LIN {X 0,Y 347.72,Z 388.171,A -85,B 0,C 180,E1 -13726.687,E2 -13726.687} C_VEL
LIN {X 0,Y 347.741,Z 388.168,A -85,B 0,C 180,E1 -13730.174,E2 -13730.174} C_VEL
LIN {X 0,Y 347.757,Z 388.167,A -85,B 0,C 180,E1 -13732.681,E2 -13732.681} C_VEL
LIN {X 0,Y 347.743,Z 388.169,A -85,B 0,C 180,E1 -13735.958,E2 -13735.958} C_VEL
LIN {X 0,Y 347.838,Z 388.219,A -85,B 0,C 180,E1 -13739.799,E2 -13739.799} C_VEL
LIN {X 0,Y 350.158,Z 399.265,A -85,B 0,C 180,E1 -13742.833,E2 -13742.833} C_VEL
LIN {X 0,Y 351.631,Z 408.22,A -85,B 0,C 180,E1 -13745.185,E2 -13745.185} C_VEL
LIN {X 0,Y 351.614,Z 408.733,A -85,B 0,C 180,E1 -13745.302,E2 -13745.302} C_VEL
LIN {X 0,Y 355.783,Z 429.347,A -85,B 0,C 180,E1 -13746.384,E2 -13746.384} C_VEL
LIN {X 0,Y 358.162,Z 444.826,A -85,B 0,C 180,E1 -13747.086,E2 -13747.086} C_VEL
LIN {X 0,Y 359.103,Z 454.426,A -85,B 0,C 180,E1 -13747.462,E2 -13747.462} C_VEL
LIN {X 0,Y 356.443,Z 527.667,A -85,B 0,C 180,E1 -13749.403,E2 -13749.403} C_VEL
LIN {X 0,Y 355.433,Z 541.2,A -85,B 0,C 180,E1 -13749.983,E2 -13749.983} C_VEL
LIN {X 0,Y 354.327,Z 553.435,A -85,B 0,C 180,E1 -13750.748,E2 -13750.748} C_VEL
LIN {X 0,Y 353.054,Z 565.374,A -85,B 0,C 180,E1 -13751.73,E2 -13751.73} C_VEL
LIN {X 0,Y 351.787,Z 576.175,A -85,B 0,C 180,E1 -13752.864,E2 -13752.864} C_VEL
LIN {X 0,Y 350.439,Z 586.967,A -85,B 0,C 180,E1 -13754.288,E2 -13754.288} C_VEL
LIN {X 0,Y 349.396,Z 595.866,A -85,B 0,C 180,E1 -13755.737,E2 -13755.737} C_VEL
LIN {X 0,Y 348.24,Z 604.478,A -85,B 0,C 180,E1 -13757.472,E2 -13757.472} C_VEL
LIN {X 0,Y 347.356,Z 611.404,A -85,B 0,C 180,E1 -13759.215,E2 -13759.215} C_VEL
LIN {X 0,Y 346.698,Z 617.747,A -85,B 0,C 180,E1 -13761.257,E2 -13761.257} C_VEL
LIN {X 0,Y 346.364,Z 621.852,A -85,B 0,C 180,E1 -13763.009,E2 -13763.009} C_VEL
LIN {X 0,Y 346.173,Z 625.978,A -85,B 0,C 180,E1 -13765.344,E2 -13765.344} C_VEL
LIN {X 0,Y 346.146,Z 627.567,A -85,B 0,C 180,E1 -13766.509,E2 -13766.509} C_VEL
LIN {X 0,Y 346.085,Z 628.723,A -85,B 0,C 180,E1 -13767.674,E2 -13767.674} C_VEL
LIN {X 0,Y 346.118,Z 629.437,A -85,B 0,C 180,E1 -13768.838,E2 -13768.838} C_VEL
LIN {X 0,Y 346.164,Z 629.755,A -85,B 0,C 180,E1 -13770.002,E2 -13770.002} C_VEL
LIN {X 0,Y 346.103,Z 629.676,A -85,B 0,C 180,E1 -13771.165,E2 -13771.165} C_VEL
LIN {X 0,Y 346.083,Z 629.185,A -85,B 0,C 180,E1 -13772.329,E2 -13772.329} C_VEL
LIN {X 0,Y 346.142,Z 628.26,A -85,B 0,C 180,E1 -13773.494,E2 -13773.494} C_VEL
LIN {X 0,Y 346.161,Z 626.933,A -85,B 0,C 180,E1 -13774.66,E2 -13774.66} C_VEL
LIN {X 0,Y 346.261,Z 624.135,A -85,B 0,C 180,E1 -13776.41,E2 -13776.41} C_VEL
LIN {X 0,Y 346.568,Z 620.305,A -85,B 0,C 180,E1 -13778.162,E2 -13778.162} C_VEL
LIN {X 0,Y 347.043,Z 615.354,A -85,B 0,C 180,E1 -13779.913,E2 -13779.913} C_VEL
LIN {X 0,Y 347.727,Z 609.133,A -85,B 0,C 180,E1 -13781.662,E2 -13781.662} C_VEL
LIN {X 0,Y 348.808,Z 601.409,A -85,B 0,C 180,E1 -13783.399,E2 -13783.399} C_VEL
LIN {X 0,Y 349.843,Z 593.517,A -85,B 0,C 180,E1 -13784.842,E2 -13784.842} C_VEL
LIN {X 0,Y 350.944,Z 583.905,A -85,B 0,C 180,E1 -13786.283,E2 -13786.283} C_VEL
LIN {X 0,Y 352.227,Z 573.271,A -85,B 0,C 180,E1 -13787.567,E2 -13787.567} C_VEL
LIN {X 0,Y 353.609,Z 561.389,A -85,B 0,C 180,E1 -13788.694,E2 -13788.694} C_VEL
LIN {X 0,Y 354.715,Z 548.741,A -85,B 0,C 180,E1 -13789.609,E2 -13789.609} C_VEL
LIN {X 0,Y 355.742,Z 536.184,A -85,B 0,C 180,E1 -13790.265,E2 -13790.265} C_VEL
LIN {X 0,Y 356.474,Z 523.056,A -85,B 0,C 180,E1 -13790.712,E2 -13790.712} C_VEL
LIN {X 0,Y 357.988,Z 452.327,A -85,B 0,C 180,E1 -13792.264,E2 -13792.264} C_VEL
LIN {X 0,Y 354.472,Z 430.592,A -85,B 0,C 180,E1 -13793.053,E2 -13793.053} C_VEL
LIN {X 0,Y 351.716,Z 416.728,A -85,B 0,C 180,E1 -13793.635,E2 -13793.635} C_VEL
LIN {X 0,Y 352.39,Z 410.952,A -85,B 0,C 180,E1 -13795.077,E2 -13795.077} C_VEL
LIN {X 0,Y 351.496,Z 404.927,A -85,B 0,C 180,E1 -13796.737,E2 -13796.737} C_VEL
LIN {X 0,Y 349.55,Z 395.513,A -85,B 0,C 180,E1 -13799.471,E2 -13799.471} C_VEL
LIN {X 0,Y 347.759,Z 388.171,A -85,B 0,C 180,E1 -13801.755,E2 -13801.755} C_VEL
LIN {X 0,Y 347.794,Z 388.165,A -85,B 0,C 180,E1 -13805.876,E2 -13805.876} C_VEL
LIN {X 0,Y 347.757,Z 388.171,A -85,B 0,C 180,E1 -13808.793,E2 -13808.793} C_VEL
LIN {X 0,Y 347.756,Z 388.17,A -85,B 0,C 180,E1 -13811.831,E2 -13811.831} C_VEL
LIN {X 0,Y 347.711,Z 388.173,A -85,B 0,C 180,E1 -13815.027,E2 -13815.027} C_VEL
LIN {X 0,Y 347.756,Z 388.167,A -85,B 0,C 180,E1 -13818.398,E2 -13818.398} C_VEL
LIN {X 0,Y 347.779,Z 388.163,A -85,B 0,C 180,E1 -13822.012,E2 -13822.012} C_VEL
LIN {X 0,Y 347.75,Z 388.163,A -85,B 0,C 180,E1 -13825.537,E2 -13825.537} C_VEL
LIN {X 0,Y 347.751,Z 388.168,A -85,B 0,C 180,E1 -13828.301,E2 -13828.301} C_VEL
LIN {X 0,Y 347.785,Z 388.164,A -85,B 0,C 180,E1 -13830.988,E2 -13830.988} C_VEL
LIN {X 0,Y 347.837,Z 388.149,A -85,B 0,C 180,E1 -13833.608,E2 -13833.608} C_VEL
LIN {X 0,Y 347.795,Z 388.162,A -85,B 0,C 180,E1 -13836.162,E2 -13836.162} C_VEL
LIN {X 0,Y 347.819,Z 388.159,A -85,B 0,C 180,E1 -13839.91,E2 -13839.91} C_VEL
LIN {X 0,Y 347.873,Z 388.148,A -85,B 0,C 180,E1 -13842.36,E2 -13842.36} C_VEL
LIN {X 0,Y 347.904,Z 388.14,A -85,B 0,C 180,E1 -13845.971,E2 -13845.971} C_VEL
LIN {X 0,Y 347.935,Z 388.136,A -85,B 0,C 180,E1 -13849.526,E2 -13849.526} C_VEL
LIN {X 0,Y 348.081,Z 388.128,A -85,B 0,C 180,E1 -13851.875,E2 -13851.875} C_VEL
LIN {X 0,Y 348.074,Z 388.123,A -85,B 0,C 180,E1 -13854.206,E2 -13854.206} C_VEL
LIN {X 0,Y 348.212,Z 388.103,A -85,B 0,C 180,E1 -13857.687,E2 -13857.687} C_VEL
LIN {X 0,Y 348.332,Z 388.092,A -85,B 0,C 180,E1 -13860,E2 -13860} C_VEL
LIN {X 0,Y 348.213,Z 388.111,A -85,B 0,C 180,E1 -13862.314,E2 -13862.314} C_VEL
LIN {X 0,Y 348.113,Z 388.118,A -85,B 0,C 180,E1 -13866.958,E2 -13866.958} C_VEL
LIN {X 0,Y 347.974,Z 388.139,A -85,B 0,C 180,E1 -13869.298,E2 -13869.298} C_VEL
LIN {X 0,Y 347.897,Z 388.149,A -85,B 0,C 180,E1 -13872.839,E2 -13872.839} C_VEL
LIN {X 0,Y 347.846,Z 388.157,A -85,B 0,C 180,E1 -13876.431,E2 -13876.431} C_VEL
LIN {X 0,Y 347.863,Z 388.156,A -85,B 0,C 180,E1 -13878.86,E2 -13878.86} C_VEL
LIN {X 0,Y 347.781,Z 388.166,A -85,B 0,C 180,E1 -13882.579,E2 -13882.579} C_VEL
LIN {X 0,Y 347.829,Z 388.166,A -85,B 0,C 180,E1 -13884.238,E2 -13884.238} C_VEL
LIN {X 0,Y 350.024,Z 397.889,A -85,B 0,C 180,E1 -13887.504,E2 -13887.504} C_VEL
LIN {X 0,Y 350.495,Z 400.533,A -85,B 0,C 180,E1 -13888.353,E2 -13888.353} C_VEL
LIN {X 0,Y 355.561,Z 413.584,A -85,B 0,C 180,E1 -13889.086,E2 -13889.086} C_VEL
LIN {X 0,Y 358.59,Z 428.221,A -85,B 0,C 180,E1 -13889.672,E2 -13889.672} C_VEL
LIN {X 0,Y 356.597,Z 507.412,A -85,B 0,C 180,E1 -13891.413,E2 -13891.413} C_VEL
LIN {X 0,Y 355.951,Z 520.049,A -85,B 0,C 180,E1 -13891.895,E2 -13891.895} C_VEL
LIN {X 0,Y 355.055,Z 533.276,A -85,B 0,C 180,E1 -13892.642,E2 -13892.642} C_VEL
LIN {X 0,Y 353.946,Z 545.604,A -85,B 0,C 180,E1 -13893.604,E2 -13893.604} C_VEL
LIN {X 0,Y 352.773,Z 556.709,A -85,B 0,C 180,E1 -13894.721,E2 -13894.721} C_VEL
LIN {X 0,Y 351.601,Z 566.56,A -85,B 0,C 180,E1 -13895.956,E2 -13895.956} C_VEL
LIN {X 0,Y 350.493,Z 575.046,A -85,B 0,C 180,E1 -13897.256,E2 -13897.256} C_VEL
LIN {X 0,Y 349.382,Z 583.6,A -85,B 0,C 180,E1 -13898.868,E2 -13898.868} C_VEL
LIN {X 0,Y 348.401,Z 590.791,A -85,B 0,C 180,E1 -13900.543,E2 -13900.543} C_VEL
LIN {X 0,Y 347.524,Z 597.568,A -85,B 0,C 180,E1 -13902.536,E2 -13902.536} C_VEL
LIN {X 0,Y 346.932,Z 601.844,A -85,B 0,C 180,E1 -13904.154,E2 -13904.154} C_VEL
LIN {X 0,Y 346.562,Z 605.2,A -85,B 0,C 180,E1 -13905.792,E2 -13905.792} C_VEL
LIN {X 0,Y 346.141,Z 608.29,A -85,B 0,C 180,E1 -13907.929,E2 -13907.929} C_VEL
LIN {X 0,Y 345.978,Z 609.589,A -85,B 0,C 180,E1 -13909.455,E2 -13909.455} C_VEL
LIN {X 0,Y 345.904,Z 610.218,A -85,B 0,C 180,E1 -13910.959,E2 -13910.959} C_VEL
LIN {X 0,Y 345.879,Z 610.181,A -85,B 0,C 180,E1 -13912.44,E2 -13912.44} C_VEL
LIN {X 0,Y 345.94,Z 609.166,A -85,B 0,C 180,E1 -13914.354,E2 -13914.354} C_VEL
LIN {X 0,Y 346.175,Z 606.93,A -85,B 0,C 180,E1 -13916.344,E2 -13916.344} C_VEL
LIN {X 0,Y 346.537,Z 603.249,A -85,B 0,C 180,E1 -13918.407,E2 -13918.407} C_VEL
LIN {X 0,Y 346.857,Z 599.121,A -85,B 0,C 180,E1 -13920.107,E2 -13920.107} C_VEL
LIN {X 0,Y 347.444,Z 593.365,A -85,B 0,C 180,E1 -13921.945,E2 -13921.945} C_VEL
LIN {X 0,Y 348.176,Z 586.714,A -85,B 0,C 180,E1 -13923.634,E2 -13923.634} C_VEL
LIN {X 0,Y 349.022,Z 578.446,A -85,B 0,C 180,E1 -13925.33,E2 -13925.33} C_VEL
LIN {X 0,Y 350.071,Z 569.169,A -85,B 0,C 180,E1 -13926.851,E2 -13926.851} C_VEL
LIN {X 0,Y 351.212,Z 558.436,A -85,B 0,C 180,E1 -13928.271,E2 -13928.271} C_VEL
LIN {X 0,Y 352.121,Z 547.542,A -85,B 0,C 180,E1 -13929.422,E2 -13929.422} C_VEL
LIN {X 0,Y 353.153,Z 534.893,A -85,B 0,C 180,E1 -13930.452,E2 -13930.452} C_VEL
LIN {X 0,Y 353.886,Z 523.166,A -85,B 0,C 180,E1 -13931.171,E2 -13931.171} C_VEL
LIN {X 0,Y 354.534,Z 510.132,A -85,B 0,C 180,E1 -13931.726,E2 -13931.726} C_VEL
LIN {X 0,Y 354.958,Z 492.695,A -85,B 0,C 180,E1 -13932.16,E2 -13932.16} C_VEL
LIN {X 0,Y 356.276,Z 426.34,A -85,B 0,C 180,E1 -13933.571,E2 -13933.571} C_VEL
LIN {X 0,Y 352.164,Z 405.889,A -85,B 0,C 180,E1 -13934.276,E2 -13934.276} C_VEL
LIN {X 0,Y 350.017,Z 399.405,A -85,B 0,C 180,E1 -13934.569,E2 -13934.569} C_VEL
LIN {X 0,Y 347.928,Z 388.186,A -85,B 0,C 180,E1 -13937.938,E2 -13937.938} C_VEL
LIN {X 0,Y 348.027,Z 388.131,A -85,B 0,C 180,E1 -13941.872,E2 -13941.872} C_VEL
LIN {X 0,Y 348.055,Z 388.13,A -85,B 0,C 180,E1 -13944.204,E2 -13944.204} C_VEL
LIN {X 0,Y 348.21,Z 388.108,A -85,B 0,C 180,E1 -13947.685,E2 -13947.685} C_VEL
LIN {X 0,Y 348.348,Z 388.093,A -85,B 0,C 180,E1 -13949.998,E2 -13949.998} C_VEL
LIN {X 0,Y 348.211,Z 388.113,A -85,B 0,C 180,E1 -13952.312,E2 -13952.312} C_VEL
LIN {X 0,Y 348.109,Z 388.12,A -85,B 0,C 180,E1 -13956.956,E2 -13956.956} C_VEL
LIN {X 0,Y 347.969,Z 388.137,A -85,B 0,C 180,E1 -13959.297,E2 -13959.297} C_VEL
LIN {X 0,Y 347.891,Z 388.147,A -85,B 0,C 180,E1 -13962.838,E2 -13962.838} C_VEL
LIN {X 0,Y 347.842,Z 388.155,A -85,B 0,C 180,E1 -13966.43,E2 -13966.43} C_VEL
LIN {X 0,Y 347.817,Z 388.156,A -85,B 0,C 180,E1 -13969.381,E2 -13969.381} C_VEL
LIN {X 0,Y 347.123,Z 388.247,A -85,B 0,C 180,E1 -13970.346,E2 -13970.346} C_VEL
LIN {X 0,Y 344.256,Z 388.606,A -85,B 0,C 180,E1 -13971.917,E2 -13971.917} C_VEL
LIN {X 0,Y 341.85,Z 388.905,A -85,B 0,C 180,E1 -13973.188,E2 -13973.188} C_VEL
LIN {X 0,Y 340.83,Z 389.03,A -85,B 0,C 180,E1 -13974.172,E2 -13974.172} C_VEL
LIN {X 0,Y 340.753,Z 389.037,A -85,B 0,C 180,E1 -13974.505,E2 -13974.505} C_VEL
LIN {X 0,Y 340.778,Z 389.036,A -85,B 0,C 180,E1 -13977.525,E2 -13977.525} C_VEL
LIN {X 0,Y 340.714,Z 389.041,A -85,B 0,C 180,E1 -13981.041,E2 -13981.041} C_VEL
LIN {X 0,Y 340.715,Z 389.043,A -85,B 0,C 180,E1 -13985.277,E2 -13985.277} C_VEL
LIN {X 0,Y 340.715,Z 389.041,A -85,B 0,C 180,E1 -13988.386,E2 -13988.386} C_VEL
LIN {X 0,Y 340.728,Z 389.041,A -85,B 0,C 180,E1 -13992.05,E2 -13992.05} C_VEL
LIN {X 0,Y 340.751,Z 389.142,A -85,B 0,C 180,E1 -13993.651,E2 -13993.651} C_VEL
LIN {X 0,Y 342.514,Z 397.857,A -85,B 0,C 180,E1 -13995.733,E2 -13995.733} C_VEL
LIN {X 0,Y 344.996,Z 407.303,A -85,B 0,C 180,E1 -13996.109,E2 -13996.109} C_VEL
LIN {X 0,Y 348.332,Z 426.928,A -85,B 0,C 180,E1 -13996.786,E2 -13996.786} C_VEL
LIN {X 0,Y 346.221,Z 507.298,A -85,B 0,C 180,E1 -13998.782,E2 -13998.782} C_VEL
LIN {X 0,Y 345.703,Z 520.636,A -85,B 0,C 180,E1 -13999.342,E2 -13999.342} C_VEL
LIN {X 0,Y 344.889,Z 534.013,A -85,B 0,C 180,E1 -14000.162,E2 -14000.162} C_VEL
LIN {X 0,Y 344.107,Z 545.469,A -85,B 0,C 180,E1 -14001.094,E2 -14001.094} C_VEL
LIN {X 0,Y 343.207,Z 556.587,A -85,B 0,C 180,E1 -14002.25,E2 -14002.25} C_VEL
LIN {X 0,Y 342.276,Z 567.32,A -85,B 0,C 180,E1 -14003.637,E2 -14003.637} C_VEL
LIN {X 0,Y 341.384,Z 576.974,A -85,B 0,C 180,E1 -14005.193,E2 -14005.193} C_VEL
LIN {X 0,Y 340.642,Z 585.34,A -85,B 0,C 180,E1 -14006.856,E2 -14006.856} C_VEL
LIN {X 0,Y 340.115,Z 591.566,A -85,B 0,C 180,E1 -14008.37,E2 -14008.37} C_VEL
LIN {X 0,Y 339.565,Z 598.161,A -85,B 0,C 180,E1 -14010.371,E2 -14010.371} C_VEL
LIN {X 0,Y 339.29,Z 602.813,A -85,B 0,C 180,E1 -14012.221,E2 -14012.221} C_VEL
LIN {X 0,Y 338.978,Z 606.451,A -85,B 0,C 180,E1 -14014.19,E2 -14014.19} C_VEL
LIN {X 0,Y 338.841,Z 608.553,A -85,B 0,C 180,E1 -14015.865,E2 -14015.865} C_VEL
LIN {X 0,Y 338.75,Z 610.039,A -85,B 0,C 180,E1 -14018.072,E2 -14018.072} C_VEL
LIN {X 0,Y 338.843,Z 610.196,A -85,B 0,C 180,E1 -14019.353,E2 -14019.353} C_VEL
LIN {X 0,Y 338.914,Z 609.887,A -85,B 0,C 180,E1 -14020.622,E2 -14020.622} C_VEL
LIN {X 0,Y 339.179,Z 608.649,A -85,B 0,C 180,E1 -14022.385,E2 -14022.385} C_VEL
LIN {X 0,Y 339.511,Z 606.116,A -85,B 0,C 180,E1 -14024.389,E2 -14024.389} C_VEL
LIN {X 0,Y 340.001,Z 602.542,A -85,B 0,C 180,E1 -14026.283,E2 -14026.283} C_VEL
LIN {X 0,Y 340.778,Z 597.891,A -85,B 0,C 180,E1 -14028.098,E2 -14028.098} C_VEL
LIN {X 0,Y 341.689,Z 591.642,A -85,B 0,C 180,E1 -14029.991,E2 -14029.991} C_VEL
LIN {X 0,Y 342.831,Z 584.319,A -85,B 0,C 180,E1 -14031.749,E2 -14031.749} C_VEL
LIN {X 0,Y 344.018,Z 576.597,A -85,B 0,C 180,E1 -14033.254,E2 -14033.254} C_VEL
LIN {X 0,Y 345.367,Z 566.981,A -85,B 0,C 180,E1 -14034.775,E2 -14034.775} C_VEL
LIN {X 0,Y 346.799,Z 556.812,A -85,B 0,C 180,E1 -14036.078,E2 -14036.078} C_VEL
LIN {X 0,Y 348.151,Z 545.387,A -85,B 0,C 180,E1 -14037.252,E2 -14037.252} C_VEL
LIN {X 0,Y 349.395,Z 532.56,A -85,B 0,C 180,E1 -14038.271,E2 -14038.271} C_VEL
LIN {X 0,Y 350.408,Z 519.533,A -85,B 0,C 180,E1 -14039.03,E2 -14039.03} C_VEL
LIN {X 0,Y 351.237,Z 505.365,A -85,B 0,C 180,E1 -14039.585,E2 -14039.585} C_VEL
LIN {X 0,Y 354.285,Z 429.068,A -85,B 0,C 180,E1 -14041.595,E2 -14041.595} C_VEL
LIN {X 0,Y 351.519,Z 416.043,A -85,B 0,C 180,E1 -14042.292,E2 -14042.292} C_VEL
LIN {X 0,Y 346.855,Z 405.479,A -85,B 0,C 180,E1 -14043.142,E2 -14043.142} C_VEL
LIN {X 0,Y 343.776,Z 399.199,A -85,B 0,C 180,E1 -14043.736,E2 -14043.736} C_VEL
LIN {X 0,Y 341.037,Z 389.005,A -85,B 0,C 180,E1 -14046.619,E2 -14046.619} C_VEL
LIN {X 0,Y 340.919,Z 389.02,A -85,B 0,C 180,E1 -14049.492,E2 -14049.492} C_VEL
LIN {X 0,Y 340.836,Z 389.031,A -85,B 0,C 180,E1 -14053.11,E2 -14053.11} C_VEL
LIN {X 0,Y 340.778,Z 389.037,A -85,B 0,C 180,E1 -14056.782,E2 -14056.782} C_VEL
LIN {X 0,Y 340.796,Z 389.035,A -85,B 0,C 180,E1 -14059.266,E2 -14059.266} C_VEL
LIN {X 0,Y 340.767,Z 389.036,A -85,B 0,C 180,E1 -14063.07,E2 -14063.07} C_VEL
LIN {X 0,Y 340.796,Z 389.034,A -85,B 0,C 180,E1 -14066.981,E2 -14066.981} C_VEL
LIN {X 0,Y 340.756,Z 389.039,A -85,B 0,C 180,E1 -14069.98,E2 -14069.98} C_VEL
LIN {X 0,Y 340.686,Z 389.048,A -85,B 0,C 180,E1 -14073.847,E2 -14073.847} C_VEL
LIN {X 0,Y 340.699,Z 389.046,A -85,B 0,C 180,E1 -14076.742,E2 -14076.742} C_VEL
LIN {X 0,Y 340.681,Z 389.048,A -85,B 0,C 180,E1 -14080.248,E2 -14080.248} C_VEL
LIN {X 0,Y 340.66,Z 389.05,A -85,B 0,C 180,E1 -14083.777,E2 -14083.777} C_VEL
LIN {X 0,Y 340.67,Z 389.051,A -85,B 0,C 180,E1 -14087.097,E2 -14087.097} C_VEL
LIN {X 0,Y 340.693,Z 389.047,A -85,B 0,C 180,E1 -14090.249,E2 -14090.249} C_VEL
LIN {X 0,Y 340.705,Z 389.044,A -85,B 0,C 180,E1 -14093.561,E2 -14093.561} C_VEL
LIN {X 0,Y 340.691,Z 389.048,A -85,B 0,C 180,E1 -14096.155,E2 -14096.155} C_VEL
LIN {X 0,Y 340.773,Z 389.154,A -85,B 0,C 180,E1 -14099.486,E2 -14099.486} C_VEL
LIN {X 0,Y 343.37,Z 401.381,A -85,B 0,C 180,E1 -14102.911,E2 -14102.911} C_VEL
LIN {X 0,Y 344.42,Z 407.215,A -85,B 0,C 180,E1 -14104.447,E2 -14104.447} C_VEL
LIN {X 0,Y 346.267,Z 413.478,A -85,B 0,C 180,E1 -14104.87,E2 -14104.87} C_VEL
LIN {X 0,Y 349.592,Z 430.004,A -85,B 0,C 180,E1 -14105.772,E2 -14105.772} C_VEL
LIN {X 0,Y 351.931,Z 445.044,A -85,B 0,C 180,E1 -14106.5,E2 -14106.5} C_VEL
LIN {X 0,Y 352.925,Z 455.244,A -85,B 0,C 180,E1 -14106.913,E2 -14106.913} C_VEL
LIN {X 0,Y 350.131,Z 526.949,A -85,B 0,C 180,E1 -14108.86,E2 -14108.86} C_VEL
LIN {X 0,Y 349.095,Z 540.506,A -85,B 0,C 180,E1 -14109.45,E2 -14109.45} C_VEL
LIN {X 0,Y 347.924,Z 552.831,A -85,B 0,C 180,E1 -14110.226,E2 -14110.226} C_VEL
LIN {X 0,Y 346.562,Z 564.849,A -85,B 0,C 180,E1 -14111.222,E2 -14111.222} C_VEL
LIN {X 0,Y 345.243,Z 575.728,A -85,B 0,C 180,E1 -14112.376,E2 -14112.376} C_VEL
LIN {X 0,Y 343.733,Z 586.753,A -85,B 0,C 180,E1 -14113.851,E2 -14113.851} C_VEL
LIN {X 0,Y 342.531,Z 596.263,A -85,B 0,C 180,E1 -14115.445,E2 -14115.445} C_VEL
LIN {X 0,Y 341.303,Z 604.719,A -85,B 0,C 180,E1 -14117.213,E2 -14117.213} C_VEL
LIN {X 0,Y 340.377,Z 611.576,A -85,B 0,C 180,E1 -14118.991,E2 -14118.991} C_VEL
LIN {X 0,Y 339.663,Z 617.816,A -85,B 0,C 180,E1 -14121.074,E2 -14121.074} C_VEL
LIN {X 0,Y 339.311,Z 621.854,A -85,B 0,C 180,E1 -14122.863,E2 -14122.863} C_VEL
LIN {X 0,Y 339.078,Z 625.706,A -85,B 0,C 180,E1 -14125.246,E2 -14125.246} C_VEL
LIN {X 0,Y 339.07,Z 627.31,A -85,B 0,C 180,E1 -14126.437,E2 -14126.437} C_VEL
LIN {X 0,Y 338.999,Z 628.489,A -85,B 0,C 180,E1 -14127.625,E2 -14127.625} C_VEL
LIN {X 0,Y 339.02,Z 629.217,A -85,B 0,C 180,E1 -14128.814,E2 -14128.814} C_VEL
LIN {X 0,Y 339.067,Z 629.547,A -85,B 0,C 180,E1 -14130.002,E2 -14130.002} C_VEL
LIN {X 0,Y 339.006,Z 629.48,A -85,B 0,C 180,E1 -14131.189,E2 -14131.189} C_VEL
LIN {X 0,Y 338.998,Z 629.011,A -85,B 0,C 180,E1 -14132.378,E2 -14132.378} C_VEL
LIN {X 0,Y 339.066,Z 628.1,A -85,B 0,C 180,E1 -14133.567,E2 -14133.567} C_VEL
LIN {X 0,Y 339.112,Z 625.216,A -85,B 0,C 180,E1 -14135.852,E2 -14135.852} C_VEL
LIN {X 0,Y 339.401,Z 621.617,A -85,B 0,C 180,E1 -14137.737,E2 -14137.737} C_VEL
LIN {X 0,Y 339.827,Z 617.086,A -85,B 0,C 180,E1 -14139.525,E2 -14139.525} C_VEL
LIN {X 0,Y 340.511,Z 611.351,A -85,B 0,C 180,E1 -14141.309,E2 -14141.309} C_VEL
LIN {X 0,Y 341.525,Z 604.174,A -85,B 0,C 180,E1 -14143.084,E2 -14143.084} C_VEL
LIN {X 0,Y 342.761,Z 595.245,A -85,B 0,C 180,E1 -14144.852,E2 -14144.852} C_VEL
LIN {X 0,Y 343.995,Z 585.259,A -85,B 0,C 180,E1 -14146.447,E2 -14146.447} C_VEL
LIN {X 0,Y 345.339,Z 574.762,A -85,B 0,C 180,E1 -14147.776,E2 -14147.776} C_VEL
LIN {X 0,Y 346.737,Z 563.351,A -85,B 0,C 180,E1 -14148.925,E2 -14148.925} C_VEL
LIN {X 0,Y 347.932,Z 551.525,A -85,B 0,C 180,E1 -14149.854,E2 -14149.854} C_VEL
LIN {X 0,Y 348.999,Z 538.551,A -85,B 0,C 180,E1 -14150.598,E2 -14150.598} C_VEL
LIN {X 0,Y 349.908,Z 524.861,A -85,B 0,C 180,E1 -14151.119,E2 -14151.119} C_VEL
LIN {X 0,Y 351.573,Z 453.595,A -85,B 0,C 180,E1 -14152.724,E2 -14152.724} C_VEL
LIN {X 0,Y 348.302,Z 432.882,A -85,B 0,C 180,E1 -14153.491,E2 -14153.491} C_VEL
LIN {X 0,Y 345,Z 416.504,A -85,B 0,C 180,E1 -14154.204,E2 -14154.204} C_VEL
LIN {X 0,Y 345.509,Z 412.267,A -85,B 0,C 180,E1 -14155.289,E2 -14155.289} C_VEL
LIN {X 0,Y 344.128,Z 403.871,A -85,B 0,C 180,E1 -14157.687,E2 -14157.687} C_VEL
LIN {X 0,Y 342.167,Z 394.993,A -85,B 0,C 180,E1 -14160.382,E2 -14160.382} C_VEL
LIN {X 0,Y 340.684,Z 389.052,A -85,B 0,C 180,E1 -14162.325,E2 -14162.325} C_VEL
LIN {X 0,Y 340.723,Z 389.044,A -85,B 0,C 180,E1 -14165.28,E2 -14165.28} C_VEL
LIN {X 0,Y 340.715,Z 389.047,A -85,B 0,C 180,E1 -14168.387,E2 -14168.387} C_VEL
LIN {X 0,Y 340.704,Z 389.048,A -85,B 0,C 180,E1 -14172.046,E2 -14172.046} C_VEL
LIN {X 0,Y 340.657,Z 389.053,A -85,B 0,C 180,E1 -14176.228,E2 -14176.228} C_VEL
LIN {X 0,Y 340.693,Z 389.041,A -85,B 0,C 180,E1 -14179.754,E2 -14179.754} C_VEL
LIN {X 0,Y 340.71,Z 389.041,A -85,B 0,C 180,E1 -14183.259,E2 -14183.259} C_VEL
LIN {X 0,Y 340.698,Z 389.04,A -85,B 0,C 180,E1 -14186.154,E2 -14186.154} C_VEL
LIN {X 0,Y 340.747,Z 389.033,A -85,B 0,C 180,E1 -14190.33,E2 -14190.33} C_VEL
LIN {X 0,Y 340.809,Z 389.024,A -85,B 0,C 180,E1 -14193.02,E2 -14193.02} C_VEL
LIN {X 0,Y 340.762,Z 389.037,A -85,B 0,C 180,E1 -14195.639,E2 -14195.639} C_VEL
LIN {X 0,Y 340.759,Z 389.037,A -85,B 0,C 180,E1 -14199.475,E2 -14199.475} C_VEL
LIN {X 0,Y 340.864,Z 389.017,A -85,B 0,C 180,E1 -14201.985,E2 -14201.985} C_VEL
LIN {X 0,Y 340.876,Z 389.014,A -85,B 0,C 180,E1 -14205.705,E2 -14205.705} C_VEL
LIN {X 0,Y 340.877,Z 389.015,A -85,B 0,C 180,E1 -14209.306,E2 -14209.306} C_VEL
LIN {X 0,Y 341.082,Z 388.991,A -85,B 0,C 180,E1 -14212.898,E2 -14212.898} C_VEL
LIN {X 0,Y 341.174,Z 388.98,A -85,B 0,C 180,E1 -14217.639,E2 -14217.639} C_VEL
LIN {X 0,Y 341.282,Z 388.97,A -85,B 0,C 180,E1 -14220,E2 -14220} C_VEL
LIN {X 0,Y 341.174,Z 388.987,A -85,B 0,C 180,E1 -14222.361,E2 -14222.361} C_VEL
LIN {X 0,Y 341.082,Z 388.994,A -85,B 0,C 180,E1 -14227.102,E2 -14227.102} C_VEL
LIN {X 0,Y 340.878,Z 389.025,A -85,B 0,C 180,E1 -14230.694,E2 -14230.694} C_VEL
LIN {X 0,Y 340.87,Z 389.024,A -85,B 0,C 180,E1 -14234.325,E2 -14234.325} C_VEL
LIN {X 0,Y 340.845,Z 389.03,A -85,B 0,C 180,E1 -14238.467,E2 -14238.467} C_VEL
LIN {X 0,Y 340.761,Z 389.04,A -85,B 0,C 180,E1 -14241.857,E2 -14241.857} C_VEL
LIN {X 0,Y 340.757,Z 389.053,A -85,B 0,C 180,E1 -14243.715,E2 -14243.715} C_VEL
LIN {X 0,Y 342.797,Z 397.988,A -85,B 0,C 180,E1 -14246.811,E2 -14246.811} C_VEL
LIN {X 0,Y 343.412,Z 400.853,A -85,B 0,C 180,E1 -14247.748,E2 -14247.748} C_VEL
LIN {X 0,Y 349.277,Z 415.294,A -85,B 0,C 180,E1 -14248.619,E2 -14248.619} C_VEL
LIN {X 0,Y 352.168,Z 429.023,A -85,B 0,C 180,E1 -14249.189,E2 -14249.189} C_VEL
LIN {X 0,Y 350.081,Z 508.162,A -85,B 0,C 180,E1 -14250.969,E2 -14250.969} C_VEL
LIN {X 0,Y 349.405,Z 520.702,A -85,B 0,C 180,E1 -14251.464,E2 -14251.464} C_VEL
LIN {X 0,Y 348.563,Z 532.323,A -85,B 0,C 180,E1 -14252.129,E2 -14252.129} C_VEL
LIN {X 0,Y 347.565,Z 543.421,A -85,B 0,C 180,E1 -14252.971,E2 -14252.971} C_VEL
LIN {X 0,Y 346.416,Z 554.353,A -85,B 0,C 180,E1 -14254.036,E2 -14254.036} C_VEL
LIN {X 0,Y 345.256,Z 563.645,A -85,B 0,C 180,E1 -14255.155,E2 -14255.155} C_VEL
LIN {X 0,Y 343.903,Z 573.946,A -85,B 0,C 180,E1 -14256.693,E2 -14256.693} C_VEL
LIN {X 0,Y 342.617,Z 582.852,A -85,B 0,C 180,E1 -14258.342,E2 -14258.342} C_VEL
LIN {X 0,Y 341.565,Z 590.039,A -85,B 0,C 180,E1 -14259.998,E2 -14259.998} C_VEL
LIN {X 0,Y 340.595,Z 596.982,A -85,B 0,C 180,E1 -14262.024,E2 -14262.024} C_VEL
LIN {X 0,Y 339.84,Z 602.692,A -85,B 0,C 180,E1 -14264.219,E2 -14264.219} C_VEL
LIN {X 0,Y 339.306,Z 606.782,A -85,B 0,C 180,E1 -14266.465,E2 -14266.465} C_VEL
LIN {X 0,Y 339.017,Z 609.108,A -85,B 0,C 180,E1 -14268.441,E2 -14268.441} C_VEL
LIN {X 0,Y 338.827,Z 610.191,A -85,B 0,C 180,E1 -14270.127,E2 -14270.127} C_VEL
LIN {X 0,Y 338.757,Z 610.441,A -85,B 0,C 180,E1 -14272.033,E2 -14272.033} C_VEL
LIN {X 0,Y 338.832,Z 609.619,A -85,B 0,C 180,E1 -14273.992,E2 -14273.992} C_VEL
LIN {X 0,Y 339.028,Z 607.609,A -85,B 0,C 180,E1 -14276.017,E2 -14276.017} C_VEL
LIN {X 0,Y 339.394,Z 604.249,A -85,B 0,C 180,E1 -14278.104,E2 -14278.104} C_VEL
LIN {X 0,Y 339.826,Z 599.117,A -85,B 0,C 180,E1 -14280.298,E2 -14280.298} C_VEL
LIN {X 0,Y 340.428,Z 593.459,A -85,B 0,C 180,E1 -14282.13,E2 -14282.13} C_VEL
LIN {X 0,Y 341.283,Z 585.953,A -85,B 0,C 180,E1 -14284.048,E2 -14284.048} C_VEL
LIN {X 0,Y 342.178,Z 577.564,A -85,B 0,C 180,E1 -14285.745,E2 -14285.745} C_VEL
LIN {X 0,Y 343.254,Z 568.286,A -85,B 0,C 180,E1 -14287.263,E2 -14287.263} C_VEL
LIN {X 0,Y 344.355,Z 558.306,A -85,B 0,C 180,E1 -14288.588,E2 -14288.588} C_VEL
LIN {X 0,Y 345.305,Z 547.35,A -85,B 0,C 180,E1 -14289.756,E2 -14289.756} C_VEL
LIN {X 0,Y 346.302,Z 535.448,A -85,B 0,C 180,E1 -14290.743,E2 -14290.743} C_VEL
LIN {X 0,Y 347.123,Z 522.735,A -85,B 0,C 180,E1 -14291.537,E2 -14291.537} C_VEL
LIN {X 0,Y 347.776,Z 509.585,A -85,B 0,C 180,E1 -14292.092,E2 -14292.092} C_VEL
LIN {X 0,Y 348.242,Z 489.439,A -85,B 0,C 180,E1 -14292.587,E2 -14292.587} C_VEL
LIN {X 0,Y 349.556,Z 427.119,A -85,B 0,C 180,E1 -14293.941,E2 -14293.941} C_VEL
LIN {X 0,Y 345.605,Z 407.6,A -85,B 0,C 180,E1 -14294.631,E2 -14294.631} C_VEL
LIN {X 0,Y 342.873,Z 399.611,A -85,B 0,C 180,E1 -14295.001,E2 -14295.001} C_VEL
LIN {X 0,Y 340.881,Z 389.025,A -85,B 0,C 180,E1 -14298.289,E2 -14298.289} C_VEL
LIN {X 0,Y 340.963,Z 389.01,A -85,B 0,C 180,E1 -14301.703,E2 -14301.703} C_VEL
LIN {X 0,Y 341.03,Z 389.004,A -85,B 0,C 180,E1 -14304.084,E2 -14304.084} C_VEL
LIN {X 0,Y 341.172,Z 388.984,A -85,B 0,C 180,E1 -14307.637,E2 -14307.637} C_VEL
LIN {X 0,Y 341.299,Z 388.971,A -85,B 0,C 180,E1 -14309.998,E2 -14309.998} C_VEL
LIN {X 0,Y 341.173,Z 388.989,A -85,B 0,C 180,E1 -14312.36,E2 -14312.36} C_VEL
LIN {X 0,Y 341.078,Z 388.995,A -85,B 0,C 180,E1 -14317.1,E2 -14317.1} C_VEL
LIN {X 0,Y 340.872,Z 389.022,A -85,B 0,C 180,E1 -14320.692,E2 -14320.692} C_VEL
LIN {X 0,Y 340.864,Z 389.026,A -85,B 0,C 180,E1 -14324.323,E2 -14324.323} C_VEL
LIN {X 0,Y 340.838,Z 389.027,A -85,B 0,C 180,E1 -14328.465,E2 -14328.465} C_VEL
LIN {X 0,Y 340.719,Z 389.045,A -85,B 0,C 180,E1 -14331.841,E2 -14331.841} C_VEL
LIN {X 0,Y 340.753,Z 389.037,A -85,B 0,C 180,E1 -14334.505,E2 -14334.505} C_VEL
LIN {X 0,Y 340.097,Z 389.122,A -85,B 0,C 180,E1 -14335.492,E2 -14335.492} C_VEL
LIN {X 0,Y 337.232,Z 389.475,A -85,B 0,C 180,E1 -14337.098,E2 -14337.098} C_VEL
LIN {X 0,Y 334.801,Z 389.778,A -85,B 0,C 180,E1 -14338.398,E2 -14338.398} C_VEL
LIN {X 0,Y 333.764,Z 389.908,A -85,B 0,C 180,E1 -14339.404,E2 -14339.404} C_VEL
LIN {X 0,Y 333.684,Z 389.914,A -85,B 0,C 180,E1 -14339.745,E2 -14339.745} C_VEL
LIN {X 0,Y 333.638,Z 389.924,A -85,B 0,C 180,E1 -14343.206,E2 -14343.206} C_VEL
LIN {X 0,Y 333.663,Z 389.92,A -85,B 0,C 180,E1 -14346.831,E2 -14346.831} C_VEL
LIN {X 0,Y 333.668,Z 389.921,A -85,B 0,C 180,E1 -14349.187,E2 -14349.187} C_VEL
LIN {X 0,Y 333.706,Z 389.931,A -85,B 0,C 180,E1 -14353.411,E2 -14353.411} C_VEL
LIN {X 0,Y 335.285,Z 397.876,A -85,B 0,C 180,E1 -14355.355,E2 -14355.355} C_VEL
LIN {X 0,Y 338.24,Z 408.461,A -85,B 0,C 180,E1 -14355.801,E2 -14355.801} C_VEL
LIN {X 0,Y 341.492,Z 427.617,A -85,B 0,C 180,E1 -14356.478,E2 -14356.478} C_VEL
LIN {X 0,Y 339.315,Z 508.15,A -85,B 0,C 180,E1 -14358.536,E2 -14358.536} C_VEL
LIN {X 0,Y 338.768,Z 521.01,A -85,B 0,C 180,E1 -14359.096,E2 -14359.096} C_VEL
LIN {X 0,Y 337.934,Z 534.446,A -85,B 0,C 180,E1 -14359.94,E2 -14359.94} C_VEL
LIN {X 0,Y 337.09,Z 546.467,A -85,B 0,C 180,E1 -14360.954,E2 -14360.954} C_VEL
LIN {X 0,Y 336.171,Z 557.273,A -85,B 0,C 180,E1 -14362.112,E2 -14362.112} C_VEL
LIN {X 0,Y 335.26,Z 567.731,A -85,B 0,C 180,E1 -14363.5,E2 -14363.5} C_VEL
LIN {X 0,Y 334.348,Z 577.187,A -85,B 0,C 180,E1 -14365.059,E2 -14365.059} C_VEL
LIN {X 0,Y 333.581,Z 585.688,A -85,B 0,C 180,E1 -14366.785,E2 -14366.785} C_VEL
LIN {X 0,Y 332.974,Z 592.551,A -85,B 0,C 180,E1 -14368.507,E2 -14368.507} C_VEL
LIN {X 0,Y 332.445,Z 598.737,A -85,B 0,C 180,E1 -14370.476,E2 -14370.476} C_VEL
LIN {X 0,Y 332.143,Z 604.029,A -85,B 0,C 180,E1 -14372.706,E2 -14372.706} C_VEL
LIN {X 0,Y 331.797,Z 607.623,A -85,B 0,C 180,E1 -14374.936,E2 -14374.936} C_VEL
LIN {X 0,Y 331.707,Z 609.069,A -85,B 0,C 180,E1 -14376.261,E2 -14376.261} C_VEL
LIN {X 0,Y 331.659,Z 609.969,A -85,B 0,C 180,E1 -14377.578,E2 -14377.578} C_VEL
LIN {X 0,Y 331.7,Z 610.375,A -85,B 0,C 180,E1 -14378.888,E2 -14378.888} C_VEL
LIN {X 0,Y 331.778,Z 610.312,A -85,B 0,C 180,E1 -14380.188,E2 -14380.188} C_VEL
LIN {X 0,Y 332.067,Z 609.178,A -85,B 0,C 180,E1 -14382.243,E2 -14382.243} C_VEL
LIN {X 0,Y 332.345,Z 607.204,A -85,B 0,C 180,E1 -14384.043,E2 -14384.043} C_VEL
LIN {X 0,Y 332.908,Z 603.561,A -85,B 0,C 180,E1 -14386.184,E2 -14386.184} C_VEL
LIN {X 0,Y 333.576,Z 599.709,A -85,B 0,C 180,E1 -14387.837,E2 -14387.837} C_VEL
LIN {X 0,Y 334.464,Z 594.123,A -85,B 0,C 180,E1 -14389.711,E2 -14389.711} C_VEL
LIN {X 0,Y 335.646,Z 587.095,A -85,B 0,C 180,E1 -14391.572,E2 -14391.572} C_VEL
LIN {X 0,Y 337.097,Z 578.291,A -85,B 0,C 180,E1 -14393.415,E2 -14393.415} C_VEL
LIN {X 0,Y 338.605,Z 568.677,A -85,B 0,C 180,E1 -14395.03,E2 -14395.03} C_VEL
LIN {X 0,Y 340.155,Z 558.057,A -85,B 0,C 180,E1 -14396.446,E2 -14396.446} C_VEL
LIN {X 0,Y 341.589,Z 546.895,A -85,B 0,C 180,E1 -14397.642,E2 -14397.642} C_VEL
LIN {X 0,Y 342.93,Z 534.355,A -85,B 0,C 180,E1 -14398.679,E2 -14398.679} C_VEL
LIN {X 0,Y 344.016,Z 521.247,A -85,B 0,C 180,E1 -14399.496,E2 -14399.496} C_VEL
LIN {X 0,Y 344.916,Z 507.427,A -85,B 0,C 180,E1 -14400.075,E2 -14400.075} C_VEL
LIN {X 0,Y 348.216,Z 430.377,A -85,B 0,C 180,E1 -14402.179,E2 -14402.179} C_VEL
LIN {X 0,Y 345.768,Z 418.733,A -85,B 0,C 180,E1 -14402.821,E2 -14402.821} C_VEL
LIN {X 0,Y 340.417,Z 406.736,A -85,B 0,C 180,E1 -14403.861,E2 -14403.861} C_VEL
LIN {X 0,Y 336.502,Z 399.359,A -85,B 0,C 180,E1 -14404.644,E2 -14404.644} C_VEL
LIN {X 0,Y 334.753,Z 392.457,A -85,B 0,C 180,E1 -14406.631,E2 -14406.631} C_VEL
LIN {X 0,Y 334.022,Z 389.881,A -85,B 0,C 180,E1 -14407.404,E2 -14407.404} C_VEL
LIN {X 0,Y 333.827,Z 389.904,A -85,B 0,C 180,E1 -14410.922,E2 -14410.922} C_VEL
LIN {X 0,Y 333.798,Z 389.909,A -85,B 0,C 180,E1 -14414.635,E2 -14414.635} C_VEL
LIN {X 0,Y 333.788,Z 389.908,A -85,B 0,C 180,E1 -14418.657,E2 -14418.657} C_VEL
LIN {X 0,Y 333.724,Z 389.915,A -85,B 0,C 180,E1 -14422.276,E2 -14422.276} C_VEL
LIN {X 0,Y 333.72,Z 389.915,A -85,B 0,C 180,E1 -14425.106,E2 -14425.106} C_VEL
LIN {X 0,Y 333.713,Z 389.916,A -85,B 0,C 180,E1 -14427.812,E2 -14427.812} C_VEL
LIN {X 0,Y 333.69,Z 389.92,A -85,B 0,C 180,E1 -14430.363,E2 -14430.363} C_VEL
LIN {X 0,Y 333.665,Z 389.922,A -85,B 0,C 180,E1 -14434.66,E2 -14434.66} C_VEL
LIN {X 0,Y 333.646,Z 389.925,A -85,B 0,C 180,E1 -14437.652,E2 -14437.652} C_VEL
LIN {X 0,Y 333.639,Z 389.924,A -85,B 0,C 180,E1 -14440.769,E2 -14440.769} C_VEL
LIN {X 0,Y 333.618,Z 389.926,A -85,B 0,C 180,E1 -14444.258,E2 -14444.258} C_VEL
LIN {X 0,Y 333.636,Z 389.925,A -85,B 0,C 180,E1 -14447.62,E2 -14447.62} C_VEL
LIN {X 0,Y 333.647,Z 389.925,A -85,B 0,C 180,E1 -14451.203,E2 -14451.203} C_VEL
LIN {X 0,Y 333.671,Z 389.92,A -85,B 0,C 180,E1 -14453.863,E2 -14453.863} C_VEL
LIN {X 0,Y 333.647,Z 389.925,A -85,B 0,C 180,E1 -14457.412,E2 -14457.412} C_VEL
LIN {X 0,Y 333.689,Z 389.929,A -85,B 0,C 180,E1 -14459.114,E2 -14459.114} C_VEL
LIN {X 0,Y 336.316,Z 402.19,A -85,B 0,C 180,E1 -14462.632,E2 -14462.632} C_VEL
LIN {X 0,Y 336.799,Z 404.817,A -85,B 0,C 180,E1 -14463.332,E2 -14463.332} C_VEL
LIN {X 0,Y 337.726,Z 407.926,A -85,B 0,C 180,E1 -14463.661,E2 -14463.661} C_VEL
LIN {X 0,Y 339.449,Z 412.146,A -85,B 0,C 180,E1 -14464.022,E2 -14464.022} C_VEL
LIN {X 0,Y 341.036,Z 417.871,A -85,B 0,C 180,E1 -14464.413,E2 -14464.413} C_VEL
LIN {X 0,Y 344.621,Z 437.161,A -85,B 0,C 180,E1 -14465.478,E2 -14465.478} C_VEL
LIN {X 0,Y 346.79,Z 454.867,A -85,B 0,C 180,E1 -14466.289,E2 -14466.289} C_VEL
LIN {X 0,Y 343.89,Z 526.566,A -85,B 0,C 180,E1 -14468.3,E2 -14468.3} C_VEL
LIN {X 0,Y 342.792,Z 540.14,A -85,B 0,C 180,E1 -14468.897,E2 -14468.897} C_VEL
LIN {X 0,Y 341.772,Z 550.5,A -85,B 0,C 180,E1 -14469.54,E2 -14469.54} C_VEL
LIN {X 0,Y 340.314,Z 562.907,A -85,B 0,C 180,E1 -14470.551,E2 -14470.551} C_VEL
LIN {X 0,Y 338.881,Z 574.049,A -85,B 0,C 180,E1 -14471.721,E2 -14471.721} C_VEL
LIN {X 0,Y 337.407,Z 584.23,A -85,B 0,C 180,E1 -14473.047,E2 -14473.047} C_VEL
LIN {X 0,Y 336.099,Z 593.449,A -85,B 0,C 180,E1 -14474.539,E2 -14474.539} C_VEL
LIN {X 0,Y 334.804,Z 602.464,A -85,B 0,C 180,E1 -14476.342,E2 -14476.342} C_VEL
LIN {X 0,Y 333.637,Z 609.702,A -85,B 0,C 180,E1 -14478.15,E2 -14478.15} C_VEL
LIN {X 0,Y 332.795,Z 616.313,A -85,B 0,C 180,E1 -14480.275,E2 -14480.275} C_VEL
LIN {X 0,Y 332.351,Z 620.67,A -85,B 0,C 180,E1 -14482.101,E2 -14482.101} C_VEL
LIN {X 0,Y 332.086,Z 624.159,A -85,B 0,C 180,E1 -14484.083,E2 -14484.083} C_VEL
LIN {X 0,Y 331.995,Z 627.044,A -85,B 0,C 180,E1 -14486.36,E2 -14486.36} C_VEL
LIN {X 0,Y 331.917,Z 628.243,A -85,B 0,C 180,E1 -14487.575,E2 -14487.575} C_VEL
LIN {X 0,Y 331.925,Z 628.992,A -85,B 0,C 180,E1 -14488.788,E2 -14488.788} C_VEL
LIN {X 0,Y 331.969,Z 629.337,A -85,B 0,C 180,E1 -14490.002,E2 -14490.002} C_VEL
LIN {X 0,Y 331.912,Z 629.284,A -85,B 0,C 180,E1 -14491.215,E2 -14491.215} C_VEL
LIN {X 0,Y 331.915,Z 628.837,A -85,B 0,C 180,E1 -14492.429,E2 -14492.429} C_VEL
LIN {X 0,Y 331.969,Z 627.947,A -85,B 0,C 180,E1 -14493.643,E2 -14493.643} C_VEL
LIN {X 0,Y 332.007,Z 625.383,A -85,B 0,C 180,E1 -14495.784,E2 -14495.784} C_VEL
LIN {X 0,Y 332.359,Z 621.519,A -85,B 0,C 180,E1 -14497.902,E2 -14497.902} C_VEL
LIN {X 0,Y 332.802,Z 617.017,A -85,B 0,C 180,E1 -14499.728,E2 -14499.728} C_VEL
LIN {X 0,Y 333.512,Z 611.312,A -85,B 0,C 180,E1 -14501.55,E2 -14501.55} C_VEL
LIN {X 0,Y 334.587,Z 604.189,A -85,B 0,C 180,E1 -14503.361,E2 -14503.361} C_VEL
LIN {X 0,Y 335.871,Z 595.322,A -85,B 0,C 180,E1 -14505.164,E2 -14505.164} C_VEL
LIN {X 0,Y 337.172,Z 585.559,A -85,B 0,C 180,E1 -14506.769,E2 -14506.769} C_VEL
LIN {X 0,Y 338.6,Z 575.057,A -85,B 0,C 180,E1 -14508.142,E2 -14508.142} C_VEL
LIN {X 0,Y 340.052,Z 563.761,A -85,B 0,C 180,E1 -14509.311,E2 -14509.311} C_VEL
LIN {X 0,Y 341.289,Z 552.111,A -85,B 0,C 180,E1 -14510.257,E2 -14510.257} C_VEL
LIN {X 0,Y 342.366,Z 539.524,A -85,B 0,C 180,E1 -14511.015,E2 -14511.015} C_VEL
LIN {X 0,Y 343.41,Z 525.303,A -85,B 0,C 180,E1 -14511.578,E2 -14511.578} C_VEL
LIN {X 0,Y 345.108,Z 454.111,A -85,B 0,C 180,E1 -14513.226,E2 -14513.226} C_VEL
LIN {X 0,Y 342.023,Z 434.292,A -85,B 0,C 180,E1 -14513.985,E2 -14513.985} C_VEL
LIN {X 0,Y 338.386,Z 416.276,A -85,B 0,C 180,E1 -14514.803,E2 -14514.803} C_VEL
LIN {X 0,Y 338.538,Z 412.404,A -85,B 0,C 180,E1 -14515.848,E2 -14515.848} C_VEL
LIN {X 0,Y 336.503,Z 401.683,A -85,B 0,C 180,E1 -14519.052,E2 -14519.052} C_VEL
LIN {X 0,Y 334.173,Z 392.064,A -85,B 0,C 180,E1 -14522.15,E2 -14522.15} C_VEL
LIN {X 0,Y 333.648,Z 389.927,A -85,B 0,C 180,E1 -14522.934,E2 -14522.934} C_VEL
LIN {X 0,Y 333.681,Z 389.923,A -85,B 0,C 180,E1 -14526.14,E2 -14526.14} C_VEL
LIN {X 0,Y 333.652,Z 389.93,A -85,B 0,C 180,E1 -14529.193,E2 -14529.193} C_VEL
LIN {X 0,Y 333.638,Z 389.928,A -85,B 0,C 180,E1 -14532.501,E2 -14532.501} C_VEL
LIN {X 0,Y 333.602,Z 389.931,A -85,B 0,C 180,E1 -14535.956,E2 -14535.956} C_VEL
LIN {X 0,Y 333.653,Z 389.92,A -85,B 0,C 180,E1 -14539.316,E2 -14539.316} C_VEL
LIN {X 0,Y 333.671,Z 389.918,A -85,B 0,C 180,E1 -14543.169,E2 -14543.169} C_VEL
LIN {X 0,Y 333.68,Z 389.916,A -85,B 0,C 180,E1 -14545.342,E2 -14545.342} C_VEL
LIN {X 0,Y 333.696,Z 389.909,A -85,B 0,C 180,E1 -14549.638,E2 -14549.638} C_VEL
LIN {X 0,Y 333.746,Z 389.909,A -85,B 0,C 180,E1 -14552.401,E2 -14552.401} C_VEL
LIN {X 0,Y 333.733,Z 389.914,A -85,B 0,C 180,E1 -14555.091,E2 -14555.091} C_VEL
LIN {X 0,Y 333.692,Z 389.919,A -85,B 0,C 180,E1 -14559.02,E2 -14559.02} C_VEL
LIN {X 0,Y 333.8,Z 389.895,A -85,B 0,C 180,E1 -14561.59,E2 -14561.59} C_VEL
LIN {X 0,Y 333.815,Z 389.893,A -85,B 0,C 180,E1 -14565.577,E2 -14565.577} C_VEL
LIN {X 0,Y 333.84,Z 389.892,A -85,B 0,C 180,E1 -14569.078,E2 -14569.078} C_VEL
LIN {X 0,Y 334.032,Z 389.869,A -85,B 0,C 180,E1 -14572.748,E2 -14572.748} C_VEL
LIN {X 0,Y 333.816,Z 389.902,A -85,B 0,C 180,E1 -14575.169,E2 -14575.169} C_VEL
LIN {X 0,Y 334.112,Z 389.859,A -85,B 0,C 180,E1 -14577.589,E2 -14577.589} C_VEL
LIN {X 0,Y 334.234,Z 389.848,A -85,B 0,C 180,E1 -14580,E2 -14580} C_VEL
LIN {X 0,Y 334.112,Z 389.867,A -85,B 0,C 180,E1 -14582.411,E2 -14582.411} C_VEL
LIN {X 0,Y 334.032,Z 389.873,A -85,B 0,C 180,E1 -14587.252,E2 -14587.252} C_VEL
LIN {X 0,Y 333.841,Z 389.901,A -85,B 0,C 180,E1 -14590.922,E2 -14590.922} C_VEL
LIN {X 0,Y 333.815,Z 389.904,A -85,B 0,C 180,E1 -14594.634,E2 -14594.634} C_VEL
LIN {X 0,Y 333.804,Z 389.907,A -85,B 0,C 180,E1 -14598.655,E2 -14598.655} C_VEL
LIN {X 0,Y 333.712,Z 390.006,A -85,B 0,C 180,E1 -14603.176,E2 -14603.176} C_VEL
LIN {X 0,Y 335.602,Z 398.129,A -85,B 0,C 180,E1 -14606.09,E2 -14606.09} C_VEL
LIN {X 0,Y 336.226,Z 401.005,A -85,B 0,C 180,E1 -14607.084,E2 -14607.084} C_VEL
LIN {X 0,Y 342.776,Z 416.679,A -85,B 0,C 180,E1 -14608.096,E2 -14608.096} C_VEL
LIN {X 0,Y 345.007,Z 425.862,A -85,B 0,C 180,E1 -14608.523,E2 -14608.523} C_VEL
LIN {X 0,Y 345.754,Z 430.963,A -85,B 0,C 180,E1 -14608.715,E2 -14608.715} C_VEL
LIN {X 0,Y 343.653,Z 507.919,A -85,B 0,C 180,E1 -14610.478,E2 -14610.478} C_VEL
LIN {X 0,Y 342.961,Z 520.221,A -85,B 0,C 180,E1 -14610.962,E2 -14610.962} C_VEL
LIN {X 0,Y 342.01,Z 532.792,A -85,B 0,C 180,E1 -14611.688,E2 -14611.688} C_VEL
LIN {X 0,Y 340.865,Z 544.91,A -85,B 0,C 180,E1 -14612.641,E2 -14612.641} C_VEL
LIN {X 0,Y 339.493,Z 556.737,A -85,B 0,C 180,E1 -14613.86,E2 -14613.86} C_VEL
LIN {X 0,Y 338.125,Z 567.245,A -85,B 0,C 180,E1 -14615.225,E2 -14615.225} C_VEL
LIN {X 0,Y 336.628,Z 577.382,A -85,B 0,C 180,E1 -14616.887,E2 -14616.887} C_VEL
LIN {X 0,Y 335.311,Z 586.075,A -85,B 0,C 180,E1 -14618.67,E2 -14618.67} C_VEL
LIN {X 0,Y 334.339,Z 592.685,A -85,B 0,C 180,E1 -14620.359,E2 -14620.359} C_VEL
LIN {X 0,Y 333.387,Z 599.132,A -85,B 0,C 180,E1 -14622.452,E2 -14622.452} C_VEL
LIN {X 0,Y 332.784,Z 603.266,A -85,B 0,C 180,E1 -14624.181,E2 -14624.181} C_VEL
LIN {X 0,Y 332.323,Z 606.525,A -85,B 0,C 180,E1 -14625.975,E2 -14625.975} C_VEL
LIN {X 0,Y 331.99,Z 608.861,A -85,B 0,C 180,E1 -14627.811,E2 -14627.811} C_VEL
LIN {X 0,Y 331.771,Z 610.268,A -85,B 0,C 180,E1 -14629.694,E2 -14629.694} C_VEL
LIN {X 0,Y 331.685,Z 610.628,A -85,B 0,C 180,E1 -14632.085,E2 -14632.085} C_VEL
LIN {X 0,Y 331.706,Z 610.064,A -85,B 0,C 180,E1 -14633.623,E2 -14633.623} C_VEL
LIN {X 0,Y 331.877,Z 608.256,A -85,B 0,C 180,E1 -14635.679,E2 -14635.679} C_VEL
LIN {X 0,Y 332.229,Z 605.125,A -85,B 0,C 180,E1 -14637.797,E2 -14637.797} C_VEL
LIN {X 0,Y 332.682,Z 600.382,A -85,B 0,C 180,E1 -14640.013,E2 -14640.013} C_VEL
LIN {X 0,Y 333.294,Z 594.55,A -85,B 0,C 180,E1 -14642.018,E2 -14642.018} C_VEL
LIN {X 0,Y 334.06,Z 588.061,A -85,B 0,C 180,E1 -14643.78,E2 -14643.78} C_VEL
LIN {X 0,Y 334.932,Z 580.15,A -85,B 0,C 180,E1 -14645.516,E2 -14645.516} C_VEL
LIN {X 0,Y 336.016,Z 571.242,A -85,B 0,C 180,E1 -14647.098,E2 -14647.098} C_VEL
LIN {X 0,Y 337.116,Z 561.907,A -85,B 0,C 180,E1 -14648.441,E2 -14648.441} C_VEL
LIN {X 0,Y 338.244,Z 550.242,A -85,B 0,C 180,E1 -14649.79,E2 -14649.79} C_VEL
LIN {X 0,Y 339.315,Z 538.184,A -85,B 0,C 180,E1 -14650.877,E2 -14650.877} C_VEL
LIN {X 0,Y 340.186,Z 525.665,A -85,B 0,C 180,E1 -14651.72,E2 -14651.72} C_VEL
LIN {X 0,Y 340.853,Z 512.938,A -85,B 0,C 180,E1 -14652.332,E2 -14652.332} C_VEL
LIN {X 0,Y 341.336,Z 498.764,A -85,B 0,C 180,E1 -14652.744,E2 -14652.744} C_VEL
LIN {X 0,Y 342.873,Z 428.213,A -85,B 0,C 180,E1 -14654.308,E2 -14654.308} C_VEL
LIN {X 0,Y 339.186,Z 409.945,A -85,B 0,C 180,E1 -14654.971,E2 -14654.971} C_VEL
LIN {X 0,Y 335.718,Z 399.808,A -85,B 0,C 180,E1 -14655.449,E2 -14655.449} C_VEL
LIN {X 0,Y 333.835,Z 389.904,A -85,B 0,C 180,E1 -14658.616,E2 -14658.616} C_VEL
LIN {X 0,Y 333.97,Z 389.885,A -85,B 0,C 180,E1 -14662.745,E2 -14662.745} C_VEL
LIN {X 0,Y 333.808,Z 389.902,A -85,B 0,C 180,E1 -14665.168,E2 -14665.168} C_VEL
LIN {X 0,Y 334.109,Z 389.864,A -85,B 0,C 180,E1 -14667.587,E2 -14667.587} C_VEL
LIN {X 0,Y 334.249,Z 389.849,A -85,B 0,C 180,E1 -14669.998,E2 -14669.998} C_VEL
LIN {X 0,Y 334.11,Z 389.868,A -85,B 0,C 180,E1 -14672.41,E2 -14672.41} C_VEL
LIN {X 0,Y 334.028,Z 389.874,A -85,B 0,C 180,E1 -14677.251,E2 -14677.251} C_VEL
LIN {X 0,Y 333.835,Z 389.898,A -85,B 0,C 180,E1 -14680.92,E2 -14680.92} C_VEL
LIN {X 0,Y 333.809,Z 389.902,A -85,B 0,C 180,E1 -14684.632,E2 -14684.632} C_VEL
LIN {X 0,Y 333.797,Z 389.903,A -85,B 0,C 180,E1 -14688.654,E2 -14688.654} C_VEL
LIN {X 0,Y 333.658,Z 389.922,A -85,B 0,C 180,E1 -14692.279,E2 -14692.279} C_VEL
LIN {X 0,Y 333.734,Z 389.912,A -85,B 0,C 180,E1 -14696.244,E2 -14696.244} C_VEL
LIN {X 0,Y 333.684,Z 389.914,A -85,B 0,C 180,E1 -14699.745,E2 -14699.745} C_VEL
LIN {X 0,Y 333.014,Z 390.001,A -85,B 0,C 180,E1 -14700.753,E2 -14700.753} C_VEL
LIN {X 0,Y 330.119,Z 390.361,A -85,B 0,C 180,E1 -14702.391,E2 -14702.391} C_VEL
LIN {X 0,Y 327.686,Z 390.669,A -85,B 0,C 180,E1 -14703.718,E2 -14703.718} C_VEL
LIN {X 0,Y 326.676,Z 390.79,A -85,B 0,C 180,E1 -14704.747,E2 -14704.747} C_VEL
LIN {X 0,Y 326.613,Z 390.799,A -85,B 0,C 180,E1 -14705.095,E2 -14705.095} C_VEL
LIN {X 0,Y 326.639,Z 390.794,A -85,B 0,C 180,E1 -14708.604,E2 -14708.604} C_VEL
LIN {X 0,Y 326.66,Z 390.838,A -85,B 0,C 180,E1 -14713.191,E2 -14713.191} C_VEL
LIN {X 0,Y 328.137,Z 398.182,A -85,B 0,C 180,E1 -14714.972,E2 -14714.972} C_VEL
LIN {X 0,Y 331.464,Z 409.477,A -85,B 0,C 180,E1 -14715.473,E2 -14715.473} C_VEL
LIN {X 0,Y 334.662,Z 429.285,A -85,B 0,C 180,E1 -14716.185,E2 -14716.185} C_VEL
LIN {X 0,Y 332.419,Z 507.928,A -85,B 0,C 180,E1 -14718.243,E2 -14718.243} C_VEL
LIN {X 0,Y 331.895,Z 520.122,A -85,B 0,C 180,E1 -14718.77,E2 -14718.77} C_VEL
LIN {X 0,Y 331.11,Z 533.206,A -85,B 0,C 180,E1 -14719.588,E2 -14719.588} C_VEL
LIN {X 0,Y 330.296,Z 544.597,A -85,B 0,C 180,E1 -14720.529,E2 -14720.529} C_VEL
LIN {X 0,Y 329.311,Z 556.268,A -85,B 0,C 180,E1 -14721.763,E2 -14721.763} C_VEL
LIN {X 0,Y 328.324,Z 566.907,A -85,B 0,C 180,E1 -14723.176,E2 -14723.176} C_VEL
LIN {X 0,Y 327.491,Z 575.858,A -85,B 0,C 180,E1 -14724.632,E2 -14724.632} C_VEL
LIN {X 0,Y 326.672,Z 584.249,A -85,B 0,C 180,E1 -14726.308,E2 -14726.308} C_VEL
LIN {X 0,Y 326.01,Z 591.596,A -85,B 0,C 180,E1 -14728.118,E2 -14728.118} C_VEL
LIN {X 0,Y 325.53,Z 596.861,A -85,B 0,C 180,E1 -14729.716,E2 -14729.716} C_VEL
LIN {X 0,Y 325.157,Z 601.841,A -85,B 0,C 180,E1 -14731.607,E2 -14731.607} C_VEL
LIN {X 0,Y 324.894,Z 605.926,A -85,B 0,C 180,E1 -14733.676,E2 -14733.676} C_VEL
LIN {X 0,Y 324.658,Z 608.646,A -85,B 0,C 180,E1 -14735.713,E2 -14735.713} C_VEL
LIN {X 0,Y 324.577,Z 609.788,A -85,B 0,C 180,E1 -14737.061,E2 -14737.061} C_VEL
LIN {X 0,Y 324.587,Z 610.499,A -85,B 0,C 180,E1 -14738.592,E2 -14738.592} C_VEL
LIN {X 0,Y 324.664,Z 610.591,A -85,B 0,C 180,E1 -14739.735,E2 -14739.735} C_VEL
LIN {X 0,Y 324.948,Z 609.675,A -85,B 0,C 180,E1 -14742.101,E2 -14742.101} C_VEL
LIN {X 0,Y 325.183,Z 608.177,A -85,B 0,C 180,E1 -14743.682,E2 -14743.682} C_VEL
LIN {X 0,Y 325.477,Z 606.448,A -85,B 0,C 180,E1 -14744.982,E2 -14744.982} C_VEL
LIN {X 0,Y 326.097,Z 602.894,A -85,B 0,C 180,E1 -14746.921,E2 -14746.921} C_VEL
LIN {X 0,Y 326.985,Z 598.136,A -85,B 0,C 180,E1 -14748.846,E2 -14748.846} C_VEL
LIN {X 0,Y 328.172,Z 591.524,A -85,B 0,C 180,E1 -14750.908,E2 -14750.908} C_VEL
LIN {X 0,Y 329.396,Z 584.51,A -85,B 0,C 180,E1 -14752.645,E2 -14752.645} C_VEL
LIN {X 0,Y 330.77,Z 576.575,A -85,B 0,C 180,E1 -14754.238,E2 -14754.238} C_VEL
LIN {X 0,Y 332.474,Z 566.052,A -85,B 0,C 180,E1 -14755.932,E2 -14755.932} C_VEL
LIN {X 0,Y 334.083,Z 555.511,A -85,B 0,C 180,E1 -14757.287,E2 -14757.287} C_VEL
LIN {X 0,Y 335.617,Z 543.649,A -85,B 0,C 180,E1 -14758.5,E2 -14758.5} C_VEL
LIN {X 0,Y 336.965,Z 531.142,A -85,B 0,C 180,E1 -14759.487,E2 -14759.487} C_VEL
LIN {X 0,Y 338.155,Z 516.964,A -85,B 0,C 180,E1 -14760.296,E2 -14760.296} C_VEL
LIN {X 0,Y 338.944,Z 503.488,A -85,B 0,C 180,E1 -14760.795,E2 -14760.795} C_VEL
LIN {X 0,Y 342.226,Z 431.717,A -85,B 0,C 180,E1 -14762.785,E2 -14762.785} C_VEL
LIN {X 0,Y 340.14,Z 421.595,A -85,B 0,C 180,E1 -14763.376,E2 -14763.376} C_VEL
LIN {X 0,Y 335.053,Z 410.266,A -85,B 0,C 180,E1 -14764.398,E2 -14764.398} C_VEL
LIN {X 0,Y 329.466,Z 399.594,A -85,B 0,C 180,E1 -14765.586,E2 -14765.586} C_VEL
LIN {X 0,Y 327.832,Z 393.605,A -85,B 0,C 180,E1 -14767.39,E2 -14767.39} C_VEL
LIN {X 0,Y 326.938,Z 390.759,A -85,B 0,C 180,E1 -14768.345,E2 -14768.345} C_VEL
LIN {X 0,Y 326.728,Z 390.784,A -85,B 0,C 180,E1 -14772.421,E2 -14772.421} C_VEL
LIN {X 0,Y 326.744,Z 390.786,A -85,B 0,C 180,E1 -14774.958,E2 -14774.958} C_VEL
LIN {X 0,Y 326.753,Z 390.784,A -85,B 0,C 180,E1 -14778.855,E2 -14778.855} C_VEL
LIN {X 0,Y 326.678,Z 390.791,A -85,B 0,C 180,E1 -14782.783,E2 -14782.783} C_VEL
LIN {X 0,Y 326.677,Z 390.793,A -85,B 0,C 180,E1 -14786.858,E2 -14786.858} C_VEL
LIN {X 0,Y 326.632,Z 390.799,A -85,B 0,C 180,E1 -14790.613,E2 -14790.613} C_VEL
LIN {X 0,Y 326.6,Z 390.803,A -85,B 0,C 180,E1 -14794.02,E2 -14794.02} C_VEL
LIN {X 0,Y 326.621,Z 390.799,A -85,B 0,C 180,E1 -14797.24,E2 -14797.24} C_VEL
LIN {X 0,Y 326.57,Z 390.806,A -85,B 0,C 180,E1 -14801.133,E2 -14801.133} C_VEL
LIN {X 0,Y 326.549,Z 390.807,A -85,B 0,C 180,E1 -14804.749,E2 -14804.749} C_VEL
LIN {X 0,Y 326.57,Z 390.805,A -85,B 0,C 180,E1 -14808.156,E2 -14808.156} C_VEL
LIN {X 0,Y 326.618,Z 390.801,A -85,B 0,C 180,E1 -14811.393,E2 -14811.393} C_VEL
LIN {X 0,Y 326.615,Z 390.802,A -85,B 0,C 180,E1 -14814.853,E2 -14814.853} C_VEL
LIN {X 0,Y 326.631,Z 390.874,A -85,B 0,C 180,E1 -14818.776,E2 -14818.776} C_VEL
LIN {X 0,Y 328.984,Z 401.701,A -85,B 0,C 180,E1 -14821.969,E2 -14821.969} C_VEL
LIN {X 0,Y 330.772,Z 407.25,A -85,B 0,C 180,E1 -14822.725,E2 -14822.725} C_VEL
LIN {X 0,Y 334.588,Z 416.949,A -85,B 0,C 180,E1 -14823.592,E2 -14823.592} C_VEL
LIN {X 0,Y 337.595,Z 432.003,A -85,B 0,C 180,E1 -14824.497,E2 -14824.497} C_VEL
LIN {X 0,Y 339.836,Z 446.988,A -85,B 0,C 180,E1 -14825.286,E2 -14825.286} C_VEL
LIN {X 0,Y 340.805,Z 456.813,A -85,B 0,C 180,E1 -14825.724,E2 -14825.724} C_VEL
LIN {X 0,Y 337.693,Z 526.415,A -85,B 0,C 180,E1 -14827.72,E2 -14827.72} C_VEL
LIN {X 0,Y 336.534,Z 539.844,A -85,B 0,C 180,E1 -14828.325,E2 -14828.325} C_VEL
LIN {X 0,Y 335.212,Z 552.151,A -85,B 0,C 180,E1 -14829.121,E2 -14829.121} C_VEL
LIN {X 0,Y 333.712,Z 564.145,A -85,B 0,C 180,E1 -14830.15,E2 -14830.15} C_VEL
LIN {X 0,Y 332.206,Z 575.037,A -85,B 0,C 180,E1 -14831.34,E2 -14831.34} C_VEL
LIN {X 0,Y 330.669,Z 584.935,A -85,B 0,C 180,E1 -14832.691,E2 -14832.691} C_VEL
LIN {X 0,Y 329.282,Z 593.968,A -85,B 0,C 180,E1 -14834.211,E2 -14834.211} C_VEL
LIN {X 0,Y 327.929,Z 602.826,A -85,B 0,C 180,E1 -14836.05,E2 -14836.05} C_VEL
LIN {X 0,Y 326.688,Z 609.938,A -85,B 0,C 180,E1 -14837.894,E2 -14837.894} C_VEL
LIN {X 0,Y 325.783,Z 616.475,A -85,B 0,C 180,E1 -14840.064,E2 -14840.064} C_VEL
LIN {X 0,Y 325.302,Z 620.742,A -85,B 0,C 180,E1 -14841.929,E2 -14841.929} C_VEL
LIN {X 0,Y 325.009,Z 624.321,A -85,B 0,C 180,E1 -14844.103,E2 -14844.103} C_VEL
LIN {X 0,Y 324.837,Z 627.992,A -85,B 0,C 180,E1 -14847.522,E2 -14847.522} C_VEL
LIN {X 0,Y 324.833,Z 628.768,A -85,B 0,C 180,E1 -14848.762,E2 -14848.762} C_VEL
LIN {X 0,Y 324.874,Z 629.127,A -85,B 0,C 180,E1 -14850.002,E2 -14850.002} C_VEL
LIN {X 0,Y 324.821,Z 629.089,A -85,B 0,C 180,E1 -14851.241,E2 -14851.241} C_VEL
LIN {X 0,Y 324.834,Z 628.659,A -85,B 0,C 180,E1 -14852.482,E2 -14852.482} C_VEL
LIN {X 0,Y 324.875,Z 627.794,A -85,B 0,C 180,E1 -14853.723,E2 -14853.723} C_VEL
LIN {X 0,Y 324.91,Z 625.528,A -85,B 0,C 180,E1 -14855.727,E2 -14855.727} C_VEL
LIN {X 0,Y 325.289,Z 621.421,A -85,B 0,C 180,E1 -14858.075,E2 -14858.075} C_VEL
LIN {X 0,Y 325.791,Z 616.958,A -85,B 0,C 180,E1 -14859.939,E2 -14859.939} C_VEL
LIN {X 0,Y 326.533,Z 611.301,A -85,B 0,C 180,E1 -14861.8,E2 -14861.8} C_VEL
LIN {X 0,Y 327.662,Z 604.252,A -85,B 0,C 180,E1 -14863.648,E2 -14863.648} C_VEL
LIN {X 0,Y 328.997,Z 595.443,A -85,B 0,C 180,E1 -14865.489,E2 -14865.489} C_VEL
LIN {X 0,Y 330.399,Z 585.468,A -85,B 0,C 180,E1 -14867.167,E2 -14867.167} C_VEL
LIN {X 0,Y 331.855,Z 575.358,A -85,B 0,C 180,E1 -14868.523,E2 -14868.523} C_VEL
LIN {X 0,Y 333.371,Z 564.172,A -85,B 0,C 180,E1 -14869.714,E2 -14869.714} C_VEL
LIN {X 0,Y 334.733,Z 551.696,A -85,B 0,C 180,E1 -14870.752,E2 -14870.752} C_VEL
LIN {X 0,Y 335.918,Z 539.003,A -85,B 0,C 180,E1 -14871.519,E2 -14871.519} C_VEL
LIN {X 0,Y 336.973,Z 524.861,A -85,B 0,C 180,E1 -14872.084,E2 -14872.084} C_VEL
LIN {X 0,Y 338.766,Z 455.09,A -85,B 0,C 180,E1 -14873.736,E2 -14873.736} C_VEL
LIN {X 0,Y 335.751,Z 435.556,A -85,B 0,C 180,E1 -14874.51,E2 -14874.51} C_VEL
LIN {X 0,Y 331.737,Z 416.138,A -85,B 0,C 180,E1 -14875.406,E2 -14875.406} C_VEL
LIN {X 0,Y 331.423,Z 412.543,A -85,B 0,C 180,E1 -14876.445,E2 -14876.445} C_VEL
LIN {X 0,Y 329.586,Z 403.07,A -85,B 0,C 180,E1 -14879.371,E2 -14879.371} C_VEL
LIN {X 0,Y 327.301,Z 393.75,A -85,B 0,C 180,E1 -14882.469,E2 -14882.469} C_VEL
LIN {X 0,Y 326.608,Z 390.804,A -85,B 0,C 180,E1 -14883.496,E2 -14883.496} C_VEL
LIN {X 0,Y 326.633,Z 390.802,A -85,B 0,C 180,E1 -14887.24,E2 -14887.24} C_VEL
LIN {X 0,Y 326.584,Z 390.811,A -85,B 0,C 180,E1 -14891.132,E2 -14891.132} C_VEL
LIN {X 0,Y 326.533,Z 390.811,A -85,B 0,C 180,E1 -14894.744,E2 -14894.744} C_VEL
LIN {X 0,Y 326.582,Z 390.804,A -85,B 0,C 180,E1 -14898.155,E2 -14898.155} C_VEL
LIN {X 0,Y 326.629,Z 390.799,A -85,B 0,C 180,E1 -14901.392,E2 -14901.392} C_VEL
LIN {X 0,Y 326.625,Z 390.799,A -85,B 0,C 180,E1 -14904.852,E2 -14904.852} C_VEL
LIN {X 0,Y 326.614,Z 390.8,A -85,B 0,C 180,E1 -14907.456,E2 -14907.456} C_VEL
LIN {X 0,Y 326.654,Z 390.788,A -85,B 0,C 180,E1 -14910.34,E2 -14910.34} C_VEL
LIN {X 0,Y 326.696,Z 390.787,A -85,B 0,C 180,E1 -14914.517,E2 -14914.517} C_VEL
LIN {X 0,Y 326.655,Z 390.793,A -85,B 0,C 180,E1 -14918.546,E2 -14918.546} C_VEL
LIN {X 0,Y 326.751,Z 390.773,A -85,B 0,C 180,E1 -14921.178,E2 -14921.178} C_VEL
LIN {X 0,Y 326.77,Z 390.77,A -85,B 0,C 180,E1 -14925.433,E2 -14925.433} C_VEL
LIN {X 0,Y 326.776,Z 390.772,A -85,B 0,C 180,E1 -14928.839,E2 -14928.839} C_VEL
LIN {X 0,Y 326.986,Z 390.748,A -85,B 0,C 180,E1 -14932.591,E2 -14932.591} C_VEL
LIN {X 0,Y 326.784,Z 390.779,A -85,B 0,C 180,E1 -14935.065,E2 -14935.065} C_VEL
LIN {X 0,Y 327.052,Z 390.738,A -85,B 0,C 180,E1 -14937.537,E2 -14937.537} C_VEL
LIN {X 0,Y 327.186,Z 390.726,A -85,B 0,C 180,E1 -14940,E2 -14940} C_VEL
LIN {X 0,Y 327.052,Z 390.746,A -85,B 0,C 180,E1 -14942.463,E2 -14942.463} C_VEL
LIN {X 0,Y 326.978,Z 390.751,A -85,B 0,C 180,E1 -14946.657,E2 -14946.657} C_VEL
LIN {X 0,Y 326.821,Z 390.774,A -85,B 0,C 180,E1 -14949.906,E2 -14949.906} C_VEL
LIN {X 0,Y 326.766,Z 390.781,A -85,B 0,C 180,E1 -14953.685,E2 -14953.685} C_VEL
LIN {X 0,Y 326.706,Z 390.79,A -85,B 0,C 180,E1 -14957.528,E2 -14957.528} C_VEL
LIN {X 0,Y 326.672,Z 390.797,A -85,B 0,C 180,E1 -14960.135,E2 -14960.135} C_VEL
LIN {X 0,Y 326.661,Z 390.821,A -85,B 0,C 180,E1 -14962.554,E2 -14962.554} C_VEL
LIN {X 0,Y 328.737,Z 399.744,A -85,B 0,C 180,E1 -14965.846,E2 -14965.846} C_VEL
LIN {X 0,Y 329.093,Z 401.384,A -85,B 0,C 180,E1 -14966.405,E2 -14966.405} C_VEL
LIN {X 0,Y 336.277,Z 417.937,A -85,B 0,C 180,E1 -14967.542,E2 -14967.542} C_VEL
LIN {X 0,Y 337.872,Z 423.072,A -85,B 0,C 180,E1 -14967.822,E2 -14967.822} C_VEL
LIN {X 0,Y 339.442,Z 431.708,A -85,B 0,C 180,E1 -14968.185,E2 -14968.185} C_VEL
LIN {X 0,Y 337.203,Z 508.343,A -85,B 0,C 180,E1 -14969.985,E2 -14969.985} C_VEL
LIN {X 0,Y 336.442,Z 521.031,A -85,B 0,C 180,E1 -14970.5,E2 -14970.5} C_VEL
LIN {X 0,Y 335.405,Z 534.127,A -85,B 0,C 180,E1 -14971.288,E2 -14971.288} C_VEL
LIN {X 0,Y 334.137,Z 546.38,A -85,B 0,C 180,E1 -14972.301,E2 -14972.301} C_VEL
LIN {X 0,Y 332.736,Z 557.941,A -85,B 0,C 180,E1 -14973.539,E2 -14973.539} C_VEL
LIN {X 0,Y 331.291,Z 568.336,A -85,B 0,C 180,E1 -14974.944,E2 -14974.944} C_VEL
LIN {X 0,Y 329.745,Z 578.31,A -85,B 0,C 180,E1 -14976.64,E2 -14976.64} C_VEL
LIN {X 0,Y 328.441,Z 586.436,A -85,B 0,C 180,E1 -14978.356,E2 -14978.356} C_VEL
LIN {X 0,Y 327.391,Z 593.063,A -85,B 0,C 180,E1 -14980.091,E2 -14980.091} C_VEL
LIN {X 0,Y 326.505,Z 598.497,A -85,B 0,C 180,E1 -14981.857,E2 -14981.857} C_VEL
LIN {X 0,Y 325.883,Z 602.838,A -85,B 0,C 180,E1 -14983.639,E2 -14983.639} C_VEL
LIN {X 0,Y 325.384,Z 606.234,A -85,B 0,C 180,E1 -14985.461,E2 -14985.461} C_VEL
LIN {X 0,Y 324.882,Z 609.264,A -85,B 0,C 180,E1 -14987.884,E2 -14987.884} C_VEL
LIN {X 0,Y 324.707,Z 610.438,A -85,B 0,C 180,E1 -14989.508,E2 -14989.508} C_VEL
LIN {X 0,Y 324.594,Z 610.884,A -85,B 0,C 180,E1 -14991.212,E2 -14991.212} C_VEL
LIN {X 0,Y 324.583,Z 610.45,A -85,B 0,C 180,E1 -14993.239,E2 -14993.239} C_VEL
LIN {X 0,Y 324.769,Z 608.884,A -85,B 0,C 180,E1 -14995.318,E2 -14995.318} C_VEL
LIN {X 0,Y 325.068,Z 605.997,A -85,B 0,C 180,E1 -14997.478,E2 -14997.478} C_VEL
LIN {X 0,Y 325.544,Z 601.536,A -85,B 0,C 180,E1 -14999.717,E2 -14999.717} C_VEL
LIN {X 0,Y 326.107,Z 596.24,A -85,B 0,C 180,E1 -15001.696,E2 -15001.696} C_VEL
LIN {X 0,Y 326.819,Z 590.168,A -85,B 0,C 180,E1 -15003.485,E2 -15003.485} C_VEL
LIN {X 0,Y 327.732,Z 582.6,A -85,B 0,C 180,E1 -15005.28,E2 -15005.28} C_VEL
LIN {X 0,Y 328.726,Z 574.553,A -85,B 0,C 180,E1 -15006.827,E2 -15006.827} C_VEL
LIN {X 0,Y 329.985,Z 564.171,A -85,B 0,C 180,E1 -15008.444,E2 -15008.444} C_VEL
LIN {X 0,Y 331.041,Z 553.851,A -85,B 0,C 180,E1 -15009.74,E2 -15009.74} C_VEL
LIN {X 0,Y 332.15,Z 542.614,A -85,B 0,C 180,E1 -15010.853,E2 -15010.853} C_VEL
LIN {X 0,Y 333.033,Z 531.149,A -85,B 0,C 180,E1 -15011.74,E2 -15011.74} C_VEL
LIN {X 0,Y 333.873,Z 518.052,A -85,B 0,C 180,E1 -15012.484,E2 -15012.484} C_VEL
LIN {X 0,Y 334.397,Z 506.447,A -85,B 0,C 180,E1 -15012.926,E2 -15012.926} C_VEL
LIN {X 0,Y 336.195,Z 429.035,A -85,B 0,C 180,E1 -15014.697,E2 -15014.697} C_VEL
LIN {X 0,Y 332.793,Z 412.374,A -85,B 0,C 180,E1 -15015.319,E2 -15015.319} C_VEL
LIN {X 0,Y 328.557,Z 400.009,A -85,B 0,C 180,E1 -15015.916,E2 -15015.916} C_VEL
LIN {X 0,Y 326.8,Z 390.781,A -85,B 0,C 180,E1 -15018.917,E2 -15018.917} C_VEL
LIN {X 0,Y 326.924,Z 390.764,A -85,B 0,C 180,E1 -15022.588,E2 -15022.588} C_VEL
LIN {X 0,Y 326.775,Z 390.779,A -85,B 0,C 180,E1 -15025.063,E2 -15025.063} C_VEL
LIN {X 0,Y 327.05,Z 390.744,A -85,B 0,C 180,E1 -15027.535,E2 -15027.535} C_VEL
LIN {X 0,Y 327.201,Z 390.727,A -85,B 0,C 180,E1 -15029.998,E2 -15029.998} C_VEL
LIN {X 0,Y 327.051,Z 390.746,A -85,B 0,C 180,E1 -15032.462,E2 -15032.462} C_VEL
LIN {X 0,Y 326.999,Z 390.755,A -85,B 0,C 180,E1 -15036.167,E2 -15036.167} C_VEL
LIN {X 0,Y 326.916,Z 390.762,A -85,B 0,C 180,E1 -15038.653,E2 -15038.653} C_VEL
LIN {X 0,Y 326.736,Z 390.784,A -85,B 0,C 180,E1 -15042.419,E2 -15042.419} C_VEL
LIN {X 0,Y 326.755,Z 390.78,A -85,B 0,C 180,E1 -15044.956,E2 -15044.956} C_VEL
LIN {X 0,Y 326.732,Z 390.782,A -85,B 0,C 180,E1 -15048.836,E2 -15048.836} C_VEL
LIN {X 0,Y 326.603,Z 390.799,A -85,B 0,C 180,E1 -15052.787,E2 -15052.787} C_VEL
LIN {X 0,Y 326.688,Z 390.79,A -85,B 0,C 180,E1 -15055.482,E2 -15055.482} C_VEL
LIN {X 0,Y 326.659,Z 390.795,A -85,B 0,C 180,E1 -15059.657,E2 -15059.657} C_VEL
LIN {X 0,Y 326.62,Z 390.797,A -85,B 0,C 180,E1 -15062.946,E2 -15062.946} C_VEL
LIN {X 0,Y 326.613,Z 390.799,A -85,B 0,C 180,E1 -15065.095,E2 -15065.095} C_VEL
LIN {X 0,Y 325.988,Z 390.881,A -85,B 0,C 180,E1 -15066.124,E2 -15066.124} C_VEL
LIN {X 0,Y 323.12,Z 391.238,A -85,B 0,C 180,E1 -15067.796,E2 -15067.796} C_VEL
LIN {X 0,Y 320.659,Z 391.541,A -85,B 0,C 180,E1 -15069.152,E2 -15069.152} C_VEL
LIN {X 0,Y 319.603,Z 391.672,A -85,B 0,C 180,E1 -15070.202,E2 -15070.202} C_VEL
LIN {X 0,Y 319.518,Z 391.681,A -85,B 0,C 180,E1 -15070.558,E2 -15070.558} C_VEL
LIN {X 0,Y 319.614,Z 391.713,A -85,B 0,C 180,E1 -15072.971,E2 -15072.971} C_VEL
LIN {X 0,Y 320.847,Z 398.057,A -85,B 0,C 180,E1 -15074.555,E2 -15074.555} C_VEL
LIN {X 0,Y 324.942,Z 411.868,A -85,B 0,C 180,E1 -15075.189,E2 -15075.189} C_VEL
LIN {X 0,Y 327.84,Z 430.066,A -85,B 0,C 180,E1 -15075.857,E2 -15075.857} C_VEL
LIN {X 0,Y 325.533,Z 507.602,A -85,B 0,C 180,E1 -15077.943,E2 -15077.943} C_VEL
LIN {X 0,Y 324.988,Z 519.785,A -85,B 0,C 180,E1 -15078.474,E2 -15078.474} C_VEL
LIN {X 0,Y 324.23,Z 532.483,A -85,B 0,C 180,E1 -15079.271,E2 -15079.271} C_VEL
LIN {X 0,Y 323.316,Z 544.955,A -85,B 0,C 180,E1 -15080.317,E2 -15080.317} C_VEL
LIN {X 0,Y 322.463,Z 555.154,A -85,B 0,C 180,E1 -15081.403,E2 -15081.403} C_VEL
LIN {X 0,Y 321.404,Z 565.966,A -85,B 0,C 180,E1 -15082.838,E2 -15082.838} C_VEL
LIN {X 0,Y 320.405,Z 576.294,A -85,B 0,C 180,E1 -15084.538,E2 -15084.538} C_VEL
LIN {X 0,Y 319.593,Z 584.72,A -85,B 0,C 180,E1 -15086.271,E2 -15086.271} C_VEL
LIN {X 0,Y 318.93,Z 591.835,A -85,B 0,C 180,E1 -15088.071,E2 -15088.071} C_VEL
LIN {X 0,Y 318.314,Z 598.553,A -85,B 0,C 180,E1 -15090.213,E2 -15090.213} C_VEL
LIN {X 0,Y 317.998,Z 603.585,A -85,B 0,C 180,E1 -15092.347,E2 -15092.347} C_VEL
LIN {X 0,Y 317.799,Z 606.154,A -85,B 0,C 180,E1 -15093.75,E2 -15093.75} C_VEL
LIN {X 0,Y 317.611,Z 608.079,A -85,B 0,C 180,E1 -15095.138,E2 -15095.138} C_VEL
LIN {X 0,Y 317.491,Z 609.512,A -85,B 0,C 180,E1 -15096.518,E2 -15096.518} C_VEL
LIN {X 0,Y 317.484,Z 610.599,A -85,B 0,C 180,E1 -15098.388,E2 -15098.388} C_VEL
LIN {X 0,Y 317.649,Z 610.699,A -85,B 0,C 180,E1 -15100.617,E2 -15100.617} C_VEL
LIN {X 0,Y 317.845,Z 610.099,A -85,B 0,C 180,E1 -15101.967,E2 -15101.967} C_VEL
LIN {X 0,Y 318.048,Z 609.071,A -85,B 0,C 180,E1 -15103.306,E2 -15103.306} C_VEL
LIN {X 0,Y 318.316,Z 607.551,A -85,B 0,C 180,E1 -15104.636,E2 -15104.636} C_VEL
LIN {X 0,Y 318.922,Z 604.351,A -85,B 0,C 180,E1 -15106.633,E2 -15106.633} C_VEL
LIN {X 0,Y 319.791,Z 600.03,A -85,B 0,C 180,E1 -15108.592,E2 -15108.592} C_VEL
LIN {X 0,Y 321.027,Z 593.618,A -85,B 0,C 180,E1 -15110.796,E2 -15110.796} C_VEL
LIN {X 0,Y 322.448,Z 586.012,A -85,B 0,C 180,E1 -15112.8,E2 -15112.8} C_VEL
LIN {X 0,Y 324.167,Z 576.878,A -85,B 0,C 180,E1 -15114.713,E2 -15114.713} C_VEL
LIN {X 0,Y 325.996,Z 566.375,A -85,B 0,C 180,E1 -15116.446,E2 -15116.446} C_VEL
LIN {X 0,Y 327.719,Z 555.688,A -85,B 0,C 180,E1 -15117.849,E2 -15117.849} C_VEL
LIN {X 0,Y 329.387,Z 543.456,A -85,B 0,C 180,E1 -15119.114,E2 -15119.114} C_VEL
LIN {X 0,Y 330.767,Z 531.133,A -85,B 0,C 180,E1 -15120.093,E2 -15120.093} C_VEL
LIN {X 0,Y 332.004,Z 517.274,A -85,B 0,C 180,E1 -15120.894,E2 -15120.894} C_VEL
LIN {X 0,Y 332.896,Z 502.805,A -85,B 0,C 180,E1 -15121.436,E2 -15121.436} C_VEL
LIN {X 0,Y 336.273,Z 432.794,A -85,B 0,C 180,E1 -15123.446,E2 -15123.446} C_VEL
LIN {X 0,Y 334.619,Z 424.699,A -85,B 0,C 180,E1 -15123.933,E2 -15123.933} C_VEL
LIN {X 0,Y 329.755,Z 413.763,A -85,B 0,C 180,E1 -15124.975,E2 -15124.975} C_VEL
LIN {X 0,Y 322.482,Z 399.954,A -85,B 0,C 180,E1 -15126.57,E2 -15126.57} C_VEL
LIN {X 0,Y 320.861,Z 394.557,A -85,B 0,C 180,E1 -15128.29,E2 -15128.29} C_VEL
LIN {X 0,Y 319.802,Z 391.651,A -85,B 0,C 180,E1 -15129.311,E2 -15129.311} C_VEL
LIN {X 0,Y 319.674,Z 391.663,A -85,B 0,C 180,E1 -15132.7,E2 -15132.7} C_VEL
LIN {X 0,Y 319.689,Z 391.664,A -85,B 0,C 180,E1 -15135.296,E2 -15135.296} C_VEL
LIN {X 0,Y 319.681,Z 391.665,A -85,B 0,C 180,E1 -15139.255,E2 -15139.255} C_VEL
LIN {X 0,Y 319.629,Z 391.67,A -85,B 0,C 180,E1 -15143.315,E2 -15143.315} C_VEL
LIN {X 0,Y 319.627,Z 391.67,A -85,B 0,C 180,E1 -15146.089,E2 -15146.089} C_VEL
LIN {X 0,Y 319.581,Z 391.677,A -85,B 0,C 180,E1 -15148.934,E2 -15148.934} C_VEL
LIN {X 0,Y 319.53,Z 391.682,A -85,B 0,C 180,E1 -15151.862,E2 -15151.862} C_VEL
LIN {X 0,Y 319.572,Z 391.677,A -85,B 0,C 180,E1 -15155.544,E2 -15155.544} C_VEL
LIN {X 0,Y 319.566,Z 391.679,A -85,B 0,C 180,E1 -15158.009,E2 -15158.009} C_VEL
LIN {X 0,Y 319.544,Z 391.683,A -85,B 0,C 180,E1 -15161.604,E2 -15161.604} C_VEL
LIN {X 0,Y 319.509,Z 391.687,A -85,B 0,C 180,E1 -15165.264,E2 -15165.264} C_VEL
LIN {X 0,Y 319.522,Z 391.685,A -85,B 0,C 180,E1 -15168.713,E2 -15168.713} C_VEL
LIN {X 0,Y 319.556,Z 391.679,A -85,B 0,C 180,E1 -15172.349,E2 -15172.349} C_VEL
LIN {X 0,Y 319.556,Z 391.68,A -85,B 0,C 180,E1 -15175.125,E2 -15175.125} C_VEL
LIN {X 0,Y 319.607,Z 391.848,A -85,B 0,C 180,E1 -15178.448,E2 -15178.448} C_VEL
LIN {X 0,Y 320.995,Z 398.295,A -85,B 0,C 180,E1 -15180.37,E2 -15180.37} C_VEL
LIN {X 0,Y 323.959,Z 407.018,A -85,B 0,C 180,E1 -15181.743,E2 -15181.743} C_VEL
LIN {X 0,Y 327.432,Z 415.378,A -85,B 0,C 180,E1 -15182.574,E2 -15182.574} C_VEL
LIN {X 0,Y 329.475,Z 420.999,A -85,B 0,C 180,E1 -15183.067,E2 -15183.067} C_VEL
LIN {X 0,Y 332.576,Z 438.506,A -85,B 0,C 180,E1 -15184.123,E2 -15184.123} C_VEL
LIN {X 0,Y 334.232,Z 450.731,A -85,B 0,C 180,E1 -15184.761,E2 -15184.761} C_VEL
LIN {X 0,Y 334.797,Z 458.478,A -85,B 0,C 180,E1 -15185.104,E2 -15185.104} C_VEL
LIN {X 0,Y 331.525,Z 526.621,A -85,B 0,C 180,E1 -15187.118,E2 -15187.118} C_VEL
LIN {X 0,Y 330.319,Z 539.895,A -85,B 0,C 180,E1 -15187.731,E2 -15187.731} C_VEL
LIN {X 0,Y 328.956,Z 552.074,A -85,B 0,C 180,E1 -15188.541,E2 -15188.541} C_VEL
LIN {X 0,Y 327.353,Z 563.968,A -85,B 0,C 180,E1 -15189.583,E2 -15189.583} C_VEL
LIN {X 0,Y 325.738,Z 574.794,A -85,B 0,C 180,E1 -15190.792,E2 -15190.792} C_VEL
LIN {X 0,Y 323.954,Z 585.661,A -85,B 0,C 180,E1 -15192.321,E2 -15192.321} C_VEL
LIN {X 0,Y 322.483,Z 594.557,A -85,B 0,C 180,E1 -15193.869,E2 -15193.869} C_VEL
LIN {X 0,Y 321.064,Z 603.232,A -85,B 0,C 180,E1 -15195.746,E2 -15195.746} C_VEL
LIN {X 0,Y 319.727,Z 610.211,A -85,B 0,C 180,E1 -15197.626,E2 -15197.626} C_VEL
LIN {X 0,Y 318.783,Z 616.633,A -85,B 0,C 180,E1 -15199.843,E2 -15199.843} C_VEL
LIN {X 0,Y 318.243,Z 620.814,A -85,B 0,C 180,E1 -15201.749,E2 -15201.749} C_VEL
LIN {X 0,Y 317.894,Z 624.562,A -85,B 0,C 180,E1 -15204.19,E2 -15204.19} C_VEL
LIN {X 0,Y 317.759,Z 627.737,A -85,B 0,C 180,E1 -15207.466,E2 -15207.466} C_VEL
LIN {X 0,Y 317.744,Z 628.544,A -85,B 0,C 180,E1 -15208.734,E2 -15208.734} C_VEL
LIN {X 0,Y 317.781,Z 628.917,A -85,B 0,C 180,E1 -15210.002,E2 -15210.002} C_VEL
LIN {X 0,Y 317.755,Z 628.48,A -85,B 0,C 180,E1 -15212.537,E2 -15212.537} C_VEL
LIN {X 0,Y 317.785,Z 627.645,A -85,B 0,C 180,E1 -15213.806,E2 -15213.806} C_VEL
LIN {X 0,Y 317.827,Z 625.643,A -85,B 0,C 180,E1 -15215.69,E2 -15215.69} C_VEL
LIN {X 0,Y 318.087,Z 622.603,A -85,B 0,C 180,E1 -15217.62,E2 -15217.62} C_VEL
LIN {X 0,Y 318.576,Z 618.546,A -85,B 0,C 180,E1 -15219.525,E2 -15219.525} C_VEL
LIN {X 0,Y 319.424,Z 612.327,A -85,B 0,C 180,E1 -15221.744,E2 -15221.744} C_VEL
LIN {X 0,Y 320.555,Z 605.555,A -85,B 0,C 180,E1 -15223.634,E2 -15223.634} C_VEL
LIN {X 0,Y 321.942,Z 597.229,A -85,B 0,C 180,E1 -15225.501,E2 -15225.501} C_VEL
LIN {X 0,Y 323.209,Z 588.594,A -85,B 0,C 180,E1 -15227.071,E2 -15227.071} C_VEL
LIN {X 0,Y 324.779,Z 578.032,A -85,B 0,C 180,E1 -15228.615,E2 -15228.615} C_VEL
LIN {X 0,Y 326.546,Z 566.198,A -85,B 0,C 180,E1 -15229.98,E2 -15229.98} C_VEL
LIN {X 0,Y 327.985,Z 554.33,A -85,B 0,C 180,E1 -15231.035,E2 -15231.035} C_VEL
LIN {X 0,Y 329.226,Z 542.104,A -85,B 0,C 180,E1 -15231.855,E2 -15231.855} C_VEL
LIN {X 0,Y 330.278,Z 529.716,A -85,B 0,C 180,E1 -15232.44,E2 -15232.44} C_VEL
LIN {X 0,Y 330.875,Z 515.33,A -85,B 0,C 180,E1 -15232.863,E2 -15232.863} C_VEL
LIN {X 0,Y 332.461,Z 456.099,A -85,B 0,C 180,E1 -15234.268,E2 -15234.268} C_VEL
LIN {X 0,Y 329.451,Z 436.615,A -85,B 0,C 180,E1 -15235.066,E2 -15235.066} C_VEL
LIN {X 0,Y 325.698,Z 418.613,A -85,B 0,C 180,E1 -15235.931,E2 -15235.931} C_VEL
LIN {X 0,Y 324.828,Z 415.839,A -85,B 0,C 180,E1 -15236.118,E2 -15236.118} C_VEL
LIN {X 0,Y 322.858,Z 405.219,A -85,B 0,C 180,E1 -15239.457,E2 -15239.457} C_VEL
LIN {X 0,Y 320.416,Z 395.208,A -85,B 0,C 180,E1 -15242.881,E2 -15242.881} C_VEL
LIN {X 0,Y 319.565,Z 391.679,A -85,B 0,C 180,E1 -15244.208,E2 -15244.208} C_VEL
LIN {X 0,Y 319.578,Z 391.682,A -85,B 0,C 180,E1 -15248.009,E2 -15248.009} C_VEL
LIN {X 0,Y 319.531,Z 391.688,A -85,B 0,C 180,E1 -15251.598,E2 -15251.598} C_VEL
LIN {X 0,Y 319.494,Z 391.689,A -85,B 0,C 180,E1 -15255.258,E2 -15255.258} C_VEL
LIN {X 0,Y 319.535,Z 391.685,A -85,B 0,C 180,E1 -15258.713,E2 -15258.713} C_VEL
LIN {X 0,Y 319.567,Z 391.676,A -85,B 0,C 180,E1 -15262.349,E2 -15262.349} C_VEL
LIN {X 0,Y 319.566,Z 391.675,A -85,B 0,C 180,E1 -15265.124,E2 -15265.124} C_VEL
LIN {X 0,Y 319.572,Z 391.67,A -85,B 0,C 180,E1 -15269.06,E2 -15269.06} C_VEL
LIN {X 0,Y 319.612,Z 391.668,A -85,B 0,C 180,E1 -15272.498,E2 -15272.498} C_VEL
LIN {X 0,Y 319.611,Z 391.672,A -85,B 0,C 180,E1 -15275.305,E2 -15275.305} C_VEL
LIN {X 0,Y 319.604,Z 391.666,A -85,B 0,C 180,E1 -15278.048,E2 -15278.048} C_VEL
LIN {X 0,Y 319.696,Z 391.653,A -85,B 0,C 180,E1 -15280.963,E2 -15280.963} C_VEL
LIN {X 0,Y 319.738,Z 391.646,A -85,B 0,C 180,E1 -15285.276,E2 -15285.276} C_VEL
LIN {X 0,Y 319.764,Z 391.645,A -85,B 0,C 180,E1 -15289.873,E2 -15289.873} C_VEL
LIN {X 0,Y 319.94,Z 391.627,A -85,B 0,C 180,E1 -15292.426,E2 -15292.426} C_VEL
LIN {X 0,Y 319.753,Z 391.655,A -85,B 0,C 180,E1 -15294.956,E2 -15294.956} C_VEL
LIN {X 0,Y 319.996,Z 391.616,A -85,B 0,C 180,E1 -15297.483,E2 -15297.483} C_VEL
LIN {X 0,Y 320.138,Z 391.603,A -85,B 0,C 180,E1 -15300,E2 -15300} C_VEL
LIN {X 0,Y 319.996,Z 391.625,A -85,B 0,C 180,E1 -15302.518,E2 -15302.518} C_VEL
LIN {X 0,Y 319.938,Z 391.627,A -85,B 0,C 180,E1 -15306.648,E2 -15306.648} C_VEL
LIN {X 0,Y 319.765,Z 391.654,A -85,B 0,C 180,E1 -15310.127,E2 -15310.127} C_VEL
LIN {X 0,Y 319.738,Z 391.657,A -85,B 0,C 180,E1 -15314.724,E2 -15314.724} C_VEL
LIN {X 0,Y 319.696,Z 391.665,A -85,B 0,C 180,E1 -15319.038,E2 -15319.038} C_VEL
LIN {X 0,Y 319.64,Z 391.796,A -85,B 0,C 180,E1 -15321.949,E2 -15321.949} C_VEL
LIN {X 0,Y 321.956,Z 401.613,A -85,B 0,C 180,E1 -15325.669,E2 -15325.669} C_VEL
LIN {X 0,Y 329.899,Z 419.453,A -85,B 0,C 180,E1 -15326.98,E2 -15326.98} C_VEL
LIN {X 0,Y 331.744,Z 425.11,A -85,B 0,C 180,E1 -15327.309,E2 -15327.309} C_VEL
LIN {X 0,Y 333.115,Z 431.753,A -85,B 0,C 180,E1 -15327.613,E2 -15327.613} C_VEL
LIN {X 0,Y 330.82,Z 508.761,A -85,B 0,C 180,E1 -15329.465,E2 -15329.465} C_VEL
LIN {X 0,Y 330.068,Z 520.988,A -85,B 0,C 180,E1 -15329.971,E2 -15329.971} C_VEL
LIN {X 0,Y 328.964,Z 534.013,A -85,B 0,C 180,E1 -15330.76,E2 -15330.76} C_VEL
LIN {X 0,Y 327.674,Z 546.11,A -85,B 0,C 180,E1 -15331.77,E2 -15331.77} C_VEL
LIN {X 0,Y 326.159,Z 557.98,A -85,B 0,C 180,E1 -15333.059,E2 -15333.059} C_VEL
LIN {X 0,Y 324.627,Z 568.462,A -85,B 0,C 180,E1 -15334.501,E2 -15334.501} C_VEL
LIN {X 0,Y 322.982,Z 578.531,A -85,B 0,C 180,E1 -15336.246,E2 -15336.246} C_VEL
LIN {X 0,Y 321.522,Z 587.097,A -85,B 0,C 180,E1 -15338.101,E2 -15338.101} C_VEL
LIN {X 0,Y 320.243,Z 594.78,A -85,B 0,C 180,E1 -15340.236,E2 -15340.236} C_VEL
LIN {X 0,Y 319.257,Z 600.801,A -85,B 0,C 180,E1 -15342.393,E2 -15342.393} C_VEL
LIN {X 0,Y 318.639,Z 604.615,A -85,B 0,C 180,E1 -15344.186,E2 -15344.186} C_VEL
LIN {X 0,Y 318.177,Z 607.397,A -85,B 0,C 180,E1 -15345.909,E2 -15345.909} C_VEL
LIN {X 0,Y 317.707,Z 610.06,A -85,B 0,C 180,E1 -15348.421,E2 -15348.421} C_VEL
LIN {X 0,Y 317.516,Z 611.051,A -85,B 0,C 180,E1 -15350.778,E2 -15350.778} C_VEL
LIN {X 0,Y 317.49,Z 610.615,A -85,B 0,C 180,E1 -15353.295,E2 -15353.295} C_VEL
LIN {X 0,Y 317.636,Z 609.43,A -85,B 0,C 180,E1 -15354.952,E2 -15354.952} C_VEL
LIN {X 0,Y 317.914,Z 606.792,A -85,B 0,C 180,E1 -15357.146,E2 -15357.146} C_VEL
LIN {X 0,Y 318.395,Z 602.5,A -85,B 0,C 180,E1 -15359.489,E2 -15359.489} C_VEL
LIN {X 0,Y 319.043,Z 596.627,A -85,B 0,C 180,E1 -15361.78,E2 -15361.78} C_VEL
LIN {X 0,Y 319.762,Z 590.731,A -85,B 0,C 180,E1 -15363.57,E2 -15363.57} C_VEL
LIN {X 0,Y 320.686,Z 583.32,A -85,B 0,C 180,E1 -15365.391,E2 -15365.391} C_VEL
LIN {X 0,Y 321.883,Z 574.103,A -85,B 0,C 180,E1 -15367.196,E2 -15367.196} C_VEL
LIN {X 0,Y 323.107,Z 564.214,A -85,B 0,C 180,E1 -15368.756,E2 -15368.756} C_VEL
LIN {X 0,Y 324.169,Z 554.237,A -85,B 0,C 180,E1 -15370.033,E2 -15370.033} C_VEL
LIN {X 0,Y 325.382,Z 542.062,A -85,B 0,C 180,E1 -15371.256,E2 -15371.256} C_VEL
LIN {X 0,Y 326.354,Z 529.723,A -85,B 0,C 180,E1 -15372.206,E2 -15372.206} C_VEL
LIN {X 0,Y 327.167,Z 517.271,A -85,B 0,C 180,E1 -15372.899,E2 -15372.899} C_VEL
LIN {X 0,Y 327.721,Z 504.233,A -85,B 0,C 180,E1 -15373.37,E2 -15373.37} C_VEL
LIN {X 0,Y 329.458,Z 429.694,A -85,B 0,C 180,E1 -15375.107,E2 -15375.107} C_VEL
LIN {X 0,Y 326.4,Z 414.625,A -85,B 0,C 180,E1 -15375.682,E2 -15375.682} C_VEL
LIN {X 0,Y 321.396,Z 400.215,A -85,B 0,C 180,E1 -15376.403,E2 -15376.403} C_VEL
LIN {X 0,Y 319.771,Z 391.655,A -85,B 0,C 180,E1 -15379.231,E2 -15379.231} C_VEL
LIN {X 0,Y 319.881,Z 391.642,A -85,B 0,C 180,E1 -15382.423,E2 -15382.423} C_VEL
LIN {X 0,Y 319.742,Z 391.655,A -85,B 0,C 180,E1 -15384.954,E2 -15384.954} C_VEL
LIN {X 0,Y 319.994,Z 391.623,A -85,B 0,C 180,E1 -15387.481,E2 -15387.481} C_VEL
LIN {X 0,Y 320.153,Z 391.605,A -85,B 0,C 180,E1 -15389.998,E2 -15389.998} C_VEL
LIN {X 0,Y 319.995,Z 391.625,A -85,B 0,C 180,E1 -15392.516,E2 -15392.516} C_VEL
LIN {X 0,Y 319.955,Z 391.631,A -85,B 0,C 180,E1 -15396.304,E2 -15396.304} C_VEL
LIN {X 0,Y 319.844,Z 391.642,A -85,B 0,C 180,E1 -15398.846,E2 -15398.846} C_VEL
LIN {X 0,Y 319.683,Z 391.661,A -85,B 0,C 180,E1 -15402.698,E2 -15402.698} C_VEL
LIN {X 0,Y 319.7,Z 391.659,A -85,B 0,C 180,E1 -15405.294,E2 -15405.294} C_VEL
LIN {X 0,Y 319.673,Z 391.661,A -85,B 0,C 180,E1 -15409.253,E2 -15409.253} C_VEL
LIN {X 0,Y 319.56,Z 391.677,A -85,B 0,C 180,E1 -15413.318,E2 -15413.318} C_VEL
LIN {X 0,Y 319.633,Z 391.668,A -85,B 0,C 180,E1 -15416.086,E2 -15416.086} C_VEL
LIN {X 0,Y 319.588,Z 391.671,A -85,B 0,C 180,E1 -15418.932,E2 -15418.932} C_VEL
LIN {X 0,Y 319.536,Z 391.684,A -85,B 0,C 180,E1 -15421.859,E2 -15421.859} C_VEL
LIN {X 0,Y 319.577,Z 391.679,A -85,B 0,C 180,E1 -15425.542,E2 -15425.542} C_VEL
LIN {X 0,Y 319.594,Z 391.674,A -85,B 0,C 180,E1 -15428.003,E2 -15428.003} C_VEL
LIN {X 0,Y 319.518,Z 391.681,A -85,B 0,C 180,E1 -15430.558,E2 -15430.558} C_VEL
LIN {X 0,Y 318.876,Z 391.922,A -85,B 0,C 180,E1 -15431.276,E2 -15431.276} C_VEL
LIN {X 0,Y 317.403,Z 392.595,A -85,B 0,C 180,E1 -15431.958,E2 -15431.958} C_VEL
LIN {X 0,Y 314.641,Z 394.637,A -85,B 0,C 180,E1 -15433.037,E2 -15433.037} C_VEL
LIN {X 0,Y 313.633,Z 396.458,A -85,B 0,C 180,E1 -15433.674,E2 -15433.674} C_VEL
LIN {X 0,Y 313.598,Z 397.919,A -85,B 0,C 180,E1 -15434.086,E2 -15434.086} C_VEL
LIN {X 0,Y 313.788,Z 398.752,A -85,B 0,C 180,E1 -15434.193,E2 -15434.193} C_VEL
LIN {X 0,Y 318.302,Z 413.851,A -85,B 0,C 180,E1 -15434.896,E2 -15434.896} C_VEL
LIN {X 0,Y 320.998,Z 430.44,A -85,B 0,C 180,E1 -15435.523,E2 -15435.523} C_VEL
LIN {X 0,Y 318.61,Z 508.597,A -85,B 0,C 180,E1 -15437.691,E2 -15437.691} C_VEL
LIN {X 0,Y 318.019,Z 520.981,A -85,B 0,C 180,E1 -15438.26,E2 -15438.26} C_VEL
LIN {X 0,Y 317.216,Z 533.74,A -85,B 0,C 180,E1 -15439.102,E2 -15439.102} C_VEL
LIN {X 0,Y 316.323,Z 545.34,A -85,B 0,C 180,E1 -15440.107,E2 -15440.107} C_VEL
LIN {X 0,Y 315.309,Z 556.823,A -85,B 0,C 180,E1 -15441.384,E2 -15441.384} C_VEL
LIN {X 0,Y 314.251,Z 567.422,A -85,B 0,C 180,E1 -15442.855,E2 -15442.855} C_VEL
LIN {X 0,Y 313.404,Z 576.136,A -85,B 0,C 180,E1 -15444.335,E2 -15444.335} C_VEL
LIN {X 0,Y 312.551,Z 584.703,A -85,B 0,C 180,E1 -15446.12,E2 -15446.12} C_VEL
LIN {X 0,Y 311.834,Z 592.072,A -85,B 0,C 180,E1 -15448.019,E2 -15448.019} C_VEL
LIN {X 0,Y 311.391,Z 597.089,A -85,B 0,C 180,E1 -15449.605,E2 -15449.605} C_VEL
LIN {X 0,Y 310.959,Z 602.644,A -85,B 0,C 180,E1 -15451.812,E2 -15451.812} C_VEL
LIN {X 0,Y 310.692,Z 606.38,A -85,B 0,C 180,E1 -15453.826,E2 -15453.826} C_VEL
LIN {X 0,Y 310.445,Z 609.08,A -85,B 0,C 180,E1 -15455.952,E2 -15455.952} C_VEL
LIN {X 0,Y 310.391,Z 610.642,A -85,B 0,C 180,E1 -15458.172,E2 -15458.172} C_VEL
LIN {X 0,Y 310.522,Z 610.992,A -85,B 0,C 180,E1 -15460.154,E2 -15460.154} C_VEL
LIN {X 0,Y 310.708,Z 610.555,A -85,B 0,C 180,E1 -15461.8,E2 -15461.8} C_VEL
LIN {X 0,Y 311.166,Z 608.562,A -85,B 0,C 180,E1 -15464.274,E2 -15464.274} C_VEL
LIN {X 0,Y 311.598,Z 606.435,A -85,B 0,C 180,E1 -15465.886,E2 -15465.886} C_VEL
LIN {X 0,Y 312.567,Z 601.815,A -85,B 0,C 180,E1 -15468.325,E2 -15468.325} C_VEL
LIN {X 0,Y 313.665,Z 596.6,A -85,B 0,C 180,E1 -15470.343,E2 -15470.343} C_VEL
LIN {X 0,Y 315.014,Z 590.098,A -85,B 0,C 180,E1 -15472.307,E2 -15472.307} C_VEL
LIN {X 0,Y 316.697,Z 581.917,A -85,B 0,C 180,E1 -15474.269,E2 -15474.269} C_VEL
LIN {X 0,Y 318.37,Z 573.148,A -85,B 0,C 180,E1 -15475.956,E2 -15475.956} C_VEL
LIN {X 0,Y 320.193,Z 563.22,A -85,B 0,C 180,E1 -15477.484,E2 -15477.484} C_VEL
LIN {X 0,Y 322.049,Z 551.585,A -85,B 0,C 180,E1 -15478.921,E2 -15478.921} C_VEL
LIN {X 0,Y 323.759,Z 539.005,A -85,B 0,C 180,E1 -15480.131,E2 -15480.131} C_VEL
LIN {X 0,Y 325.144,Z 526.773,A -85,B 0,C 180,E1 -15481.024,E2 -15481.024} C_VEL
LIN {X 0,Y 326.221,Z 514.774,A -85,B 0,C 180,E1 -15481.659,E2 -15481.659} C_VEL
LIN {X 0,Y 327.025,Z 500.893,A -85,B 0,C 180,E1 -15482.155,E2 -15482.155} C_VEL
LIN {X 0,Y 330.468,Z 434.427,A -85,B 0,C 180,E1 -15484.102,E2 -15484.102} C_VEL
LIN {X 0,Y 329.153,Z 427.729,A -85,B 0,C 180,E1 -15484.528,E2 -15484.528} C_VEL
LIN {X 0,Y 324.519,Z 417.229,A -85,B 0,C 180,E1 -15485.569,E2 -15485.569} C_VEL
LIN {X 0,Y 317.321,Z 403.71,A -85,B 0,C 180,E1 -15487.229,E2 -15487.229} C_VEL
LIN {X 0,Y 315.267,Z 399.971,A -85,B 0,C 180,E1 -15487.78,E2 -15487.78} C_VEL
LIN {X 0,Y 313.532,Z 395.008,A -85,B 0,C 180,E1 -15489.513,E2 -15489.513} C_VEL
LIN {X 0,Y 312.701,Z 392.532,A -85,B 0,C 180,E1 -15490.44,E2 -15490.44} C_VEL
LIN {X 0,Y 312.689,Z 392.538,A -85,B 0,C 180,E1 -15494.888,E2 -15494.888} C_VEL
LIN {X 0,Y 312.636,Z 392.543,A -85,B 0,C 180,E1 -15499.246,E2 -15499.246} C_VEL
LIN {X 0,Y 312.582,Z 392.547,A -85,B 0,C 180,E1 -15502.81,E2 -15502.81} C_VEL
LIN {X 0,Y 312.546,Z 392.553,A -85,B 0,C 180,E1 -15506.726,E2 -15506.726} C_VEL
LIN {X 0,Y 312.537,Z 392.554,A -85,B 0,C 180,E1 -15509.651,E2 -15509.651} C_VEL
LIN {X 0,Y 312.511,Z 392.556,A -85,B 0,C 180,E1 -15513.69,E2 -15513.69} C_VEL
LIN {X 0,Y 312.53,Z 392.554,A -85,B 0,C 180,E1 -15517.385,E2 -15517.385} C_VEL
LIN {X 0,Y 312.482,Z 392.56,A -85,B 0,C 180,E1 -15520.71,E2 -15520.71} C_VEL
LIN {X 0,Y 312.466,Z 392.561,A -85,B 0,C 180,E1 -15524.207,E2 -15524.207} C_VEL
LIN {X 0,Y 312.479,Z 392.56,A -85,B 0,C 180,E1 -15527.92,E2 -15527.92} C_VEL
LIN {X 0,Y 312.5,Z 392.558,A -85,B 0,C 180,E1 -15531.919,E2 -15531.919} C_VEL
LIN {X 0,Y 312.527,Z 392.555,A -85,B 0,C 180,E1 -15534.222,E2 -15534.222} C_VEL
LIN {X 0,Y 312.531,Z 392.634,A -85,B 0,C 180,E1 -15538.047,E2 -15538.047} C_VEL
LIN {X 0,Y 314.208,Z 398.402,A -85,B 0,C 180,E1 -15539.205,E2 -15539.205} C_VEL
LIN {X 0,Y 316.018,Z 403.59,A -85,B 0,C 180,E1 -15540.15,E2 -15540.15} C_VEL
LIN {X 0,Y 317.243,Z 407.185,A -85,B 0,C 180,E1 -15540.703,E2 -15540.703} C_VEL
LIN {X 0,Y 320.238,Z 413.798,A -85,B 0,C 180,E1 -15541.455,E2 -15541.455} C_VEL
LIN {X 0,Y 323.777,Z 422.813,A -85,B 0,C 180,E1 -15542.348,E2 -15542.348} C_VEL
LIN {X 0,Y 326.579,Z 438.176,A -85,B 0,C 180,E1 -15543.333,E2 -15543.333} C_VEL
LIN {X 0,Y 328.344,Z 451.721,A -85,B 0,C 180,E1 -15544.083,E2 -15544.083} C_VEL
LIN {X 0,Y 328.903,Z 459.278,A -85,B 0,C 180,E1 -15544.43,E2 -15544.43} C_VEL
LIN {X 0,Y 325.498,Z 526.147,A -85,B 0,C 180,E1 -15546.459,E2 -15546.459} C_VEL
LIN {X 0,Y 324.153,Z 540.03,A -85,B 0,C 180,E1 -15547.116,E2 -15547.116} C_VEL
LIN {X 0,Y 322.722,Z 552.033,A -85,B 0,C 180,E1 -15547.937,E2 -15547.937} C_VEL
LIN {X 0,Y 321.026,Z 563.9,A -85,B 0,C 180,E1 -15548.995,E2 -15548.995} C_VEL
LIN {X 0,Y 319.32,Z 574.702,A -85,B 0,C 180,E1 -15550.223,E2 -15550.223} C_VEL
LIN {X 0,Y 317.58,Z 584.544,A -85,B 0,C 180,E1 -15551.62,E2 -15551.62} C_VEL
LIN {X 0,Y 315.956,Z 593.543,A -85,B 0,C 180,E1 -15553.194,E2 -15553.194} C_VEL
LIN {X 0,Y 314.465,Z 602.375,A -85,B 0,C 180,E1 -15555.109,E2 -15555.109} C_VEL
LIN {X 0,Y 312.998,Z 609.481,A -85,B 0,C 180,E1 -15557.026,E2 -15557.026} C_VEL
LIN {X 0,Y 312.046,Z 615.172,A -85,B 0,C 180,E1 -15558.965,E2 -15558.965} C_VEL
LIN {X 0,Y 311.363,Z 619.631,A -85,B 0,C 180,E1 -15560.911,E2 -15560.911} C_VEL
LIN {X 0,Y 311.058,Z 622,A -85,B 0,C 180,E1 -15562.211,E2 -15562.211} C_VEL
LIN {X 0,Y 310.801,Z 624.76,A -85,B 0,C 180,E1 -15564.242,E2 -15564.242} C_VEL
LIN {X 0,Y 310.682,Z 627.472,A -85,B 0,C 180,E1 -15567.409,E2 -15567.409} C_VEL
LIN {X 0,Y 310.658,Z 628.312,A -85,B 0,C 180,E1 -15568.705,E2 -15568.705} C_VEL
LIN {X 0,Y 310.691,Z 628.706,A -85,B 0,C 180,E1 -15570.002,E2 -15570.002} C_VEL
LIN {X 0,Y 310.648,Z 628.7,A -85,B 0,C 180,E1 -15571.298,E2 -15571.298} C_VEL
LIN {X 0,Y 310.678,Z 628.303,A -85,B 0,C 180,E1 -15572.595,E2 -15572.595} C_VEL
LIN {X 0,Y 310.697,Z 627.501,A -85,B 0,C 180,E1 -15573.893,E2 -15573.893} C_VEL
LIN {X 0,Y 310.725,Z 625.758,A -85,B 0,C 180,E1 -15575.617,E2 -15575.617} C_VEL
LIN {X 0,Y 311.03,Z 622.512,A -85,B 0,C 180,E1 -15577.794,E2 -15577.794} C_VEL
LIN {X 0,Y 311.536,Z 618.491,A -85,B 0,C 180,E1 -15579.743,E2 -15579.743} C_VEL
LIN {X 0,Y 312.448,Z 612.329,A -85,B 0,C 180,E1 -15582.01,E2 -15582.01} C_VEL
LIN {X 0,Y 313.648,Z 605.606,A -85,B 0,C 180,E1 -15583.94,E2 -15583.94} C_VEL
LIN {X 0,Y 315.068,Z 597.471,A -85,B 0,C 180,E1 -15585.822,E2 -15585.822} C_VEL
LIN {X 0,Y 316.425,Z 588.829,A -85,B 0,C 180,E1 -15587.449,E2 -15587.449} C_VEL
LIN {X 0,Y 318.081,Z 578.389,A -85,B 0,C 180,E1 -15589.022,E2 -15589.022} C_VEL
LIN {X 0,Y 319.909,Z 566.682,A -85,B 0,C 180,E1 -15590.413,E2 -15590.413} C_VEL
LIN {X 0,Y 321.409,Z 555.063,A -85,B 0,C 180,E1 -15591.487,E2 -15591.487} C_VEL
LIN {X 0,Y 322.698,Z 543.117,A -85,B 0,C 180,E1 -15592.321,E2 -15592.321} C_VEL
LIN {X 0,Y 323.839,Z 530.335,A -85,B 0,C 180,E1 -15592.954,E2 -15592.954} C_VEL
LIN {X 0,Y 324.449,Z 517.6,A -85,B 0,C 180,E1 -15593.361,E2 -15593.361} C_VEL
LIN {X 0,Y 326.162,Z 456.855,A -85,B 0,C 180,E1 -15594.832,E2 -15594.832} C_VEL
LIN {X 0,Y 323.105,Z 436.928,A -85,B 0,C 180,E1 -15595.686,E2 -15595.686} C_VEL
LIN {X 0,Y 319.699,Z 420.84,A -85,B 0,C 180,E1 -15596.492,E2 -15596.492} C_VEL
LIN {X 0,Y 317.657,Z 415.592,A -85,B 0,C 180,E1 -15596.886,E2 -15596.886} C_VEL
LIN {X 0,Y 315.923,Z 406.605,A -85,B 0,C 180,E1 -15599.82,E2 -15599.82} C_VEL
LIN {X 0,Y 313.842,Z 397.933,A -85,B 0,C 180,E1 -15602.862,E2 -15602.862} C_VEL
LIN {X 0,Y 312.54,Z 392.556,A -85,B 0,C 180,E1 -15604.892,E2 -15604.892} C_VEL
LIN {X 0,Y 312.54,Z 392.558,A -85,B 0,C 180,E1 -15608.091,E2 -15608.091} C_VEL
LIN {X 0,Y 312.49,Z 392.563,A -85,B 0,C 180,E1 -15612.082,E2 -15612.082} C_VEL
LIN {X 0,Y 312.464,Z 392.565,A -85,B 0,C 180,E1 -15616.036,E2 -15616.036} C_VEL
LIN {X 0,Y 312.51,Z 392.551,A -85,B 0,C 180,E1 -15619.875,E2 -15619.875} C_VEL
LIN {X 0,Y 312.541,Z 392.552,A -85,B 0,C 180,E1 -15624.051,E2 -15624.051} C_VEL
LIN {X 0,Y 312.51,Z 392.557,A -85,B 0,C 180,E1 -15627.334,E2 -15627.334} C_VEL
LIN {X 0,Y 312.551,Z 392.552,A -85,B 0,C 180,E1 -15631.279,E2 -15631.279} C_VEL
LIN {X 0,Y 312.592,Z 392.546,A -85,B 0,C 180,E1 -15634.711,E2 -15634.711} C_VEL
LIN {X 0,Y 312.594,Z 392.537,A -85,B 0,C 180,E1 -15637.529,E2 -15637.529} C_VEL
LIN {X 0,Y 312.645,Z 392.53,A -85,B 0,C 180,E1 -15641.657,E2 -15641.657} C_VEL
LIN {X 0,Y 312.7,Z 392.523,A -85,B 0,C 180,E1 -15645.687,E2 -15645.687} C_VEL
LIN {X 0,Y 312.709,Z 392.523,A -85,B 0,C 180,E1 -15649.642,E2 -15649.642} C_VEL
LIN {X 0,Y 312.879,Z 392.508,A -85,B 0,C 180,E1 -15652.255,E2 -15652.255} C_VEL
LIN {X 0,Y 312.724,Z 392.531,A -85,B 0,C 180,E1 -15654.843,E2 -15654.843} C_VEL
LIN {X 0,Y 312.995,Z 392.497,A -85,B 0,C 180,E1 -15658.713,E2 -15658.713} C_VEL
LIN {X 0,Y 312.995,Z 392.493,A -85,B 0,C 180,E1 -15661.287,E2 -15661.287} C_VEL
LIN {X 0,Y 312.724,Z 392.531,A -85,B 0,C 180,E1 -15665.158,E2 -15665.158} C_VEL
LIN {X 0,Y 312.879,Z 392.511,A -85,B 0,C 180,E1 -15667.746,E2 -15667.746} C_VEL
LIN {X 0,Y 312.676,Z 392.536,A -85,B 0,C 180,E1 -15671.671,E2 -15671.671} C_VEL
LIN {X 0,Y 312.707,Z 392.533,A -85,B 0,C 180,E1 -15674.887,E2 -15674.887} C_VEL
LIN {X 0,Y 312.66,Z 392.54,A -85,B 0,C 180,E1 -15679.248,E2 -15679.248} C_VEL
LIN {X 0,Y 312.593,Z 392.644,A -85,B 0,C 180,E1 -15681.256,E2 -15681.256} C_VEL
LIN {X 0,Y 314.779,Z 401.833,A -85,B 0,C 180,E1 -15684.88,E2 -15684.88} C_VEL
LIN {X 0,Y 322.505,Z 418.552,A -85,B 0,C 180,E1 -15686.205,E2 -15686.205} C_VEL
LIN {X 0,Y 325.624,Z 426.827,A -85,B 0,C 180,E1 -15686.756,E2 -15686.756} C_VEL
LIN {X 0,Y 326.876,Z 433.71,A -85,B 0,C 180,E1 -15687.071,E2 -15687.071} C_VEL
LIN {X 0,Y 324.436,Z 509.26,A -85,B 0,C 180,E1 -15688.926,E2 -15688.926} C_VEL
LIN {X 0,Y 323.543,Z 522.507,A -85,B 0,C 180,E1 -15689.496,E2 -15689.496} C_VEL
LIN {X 0,Y 322.48,Z 534.646,A -85,B 0,C 180,E1 -15690.264,E2 -15690.264} C_VEL
LIN {X 0,Y 321.282,Z 545.576,A -85,B 0,C 180,E1 -15691.188,E2 -15691.188} C_VEL
LIN {X 0,Y 319.841,Z 556.631,A -85,B 0,C 180,E1 -15692.385,E2 -15692.385} C_VEL
LIN {X 0,Y 318.375,Z 566.304,A -85,B 0,C 180,E1 -15693.685,E2 -15693.685} C_VEL
LIN {X 0,Y 316.829,Z 575.605,A -85,B 0,C 180,E1 -15695.222,E2 -15695.222} C_VEL
LIN {X 0,Y 315.223,Z 584.35,A -85,B 0,C 180,E1 -15697.012,E2 -15697.012} C_VEL
LIN {X 0,Y 313.932,Z 591.424,A -85,B 0,C 180,E1 -15698.817,E2 -15698.817} C_VEL
LIN {X 0,Y 312.961,Z 597.17,A -85,B 0,C 180,E1 -15700.635,E2 -15700.635} C_VEL
LIN {X 0,Y 312.134,Z 601.879,A -85,B 0,C 180,E1 -15702.492,E2 -15702.492} C_VEL
LIN {X 0,Y 311.491,Z 605.605,A -85,B 0,C 180,E1 -15704.382,E2 -15704.382} C_VEL
LIN {X 0,Y 310.997,Z 608.403,A -85,B 0,C 180,E1 -15706.315,E2 -15706.315} C_VEL
LIN {X 0,Y 310.633,Z 610.286,A -85,B 0,C 180,E1 -15708.299,E2 -15708.299} C_VEL
LIN {X 0,Y 310.432,Z 611.254,A -85,B 0,C 180,E1 -15710.66,E2 -15710.66} C_VEL
LIN {X 0,Y 310.385,Z 611.144,A -85,B 0,C 180,E1 -15712.42,E2 -15712.42} C_VEL
LIN {X 0,Y 310.485,Z 609.961,A -85,B 0,C 180,E1 -15714.576,E2 -15714.576} C_VEL
LIN {X 0,Y 310.773,Z 607.541,A -85,B 0,C 180,E1 -15716.798,E2 -15716.798} C_VEL
LIN {X 0,Y 311.224,Z 603.674,A -85,B 0,C 180,E1 -15719.105,E2 -15719.105} C_VEL
LIN {X 0,Y 311.664,Z 599.535,A -85,B 0,C 180,E1 -15720.927,E2 -15720.927} C_VEL
LIN {X 0,Y 312.398,Z 593.848,A -85,B 0,C 180,E1 -15722.897,E2 -15722.897} C_VEL
LIN {X 0,Y 313.224,Z 587.108,A -85,B 0,C 180,E1 -15724.764,E2 -15724.764} C_VEL
LIN {X 0,Y 314.406,Z 578.143,A -85,B 0,C 180,E1 -15726.737,E2 -15726.737} C_VEL
LIN {X 0,Y 315.635,Z 568.64,A -85,B 0,C 180,E1 -15728.413,E2 -15728.413} C_VEL
LIN {X 0,Y 316.907,Z 558.2,A -85,B 0,C 180,E1 -15729.893,E2 -15729.893} C_VEL
LIN {X 0,Y 318.097,Z 547.028,A -85,B 0,C 180,E1 -15731.149,E2 -15731.149} C_VEL
LIN {X 0,Y 319.205,Z 534.927,A -85,B 0,C 180,E1 -15732.211,E2 -15732.211} C_VEL
LIN {X 0,Y 320.061,Z 522.893,A -85,B 0,C 180,E1 -15733.002,E2 -15733.002} C_VEL
LIN {X 0,Y 320.816,Z 509.271,A -85,B 0,C 180,E1 -15733.607,E2 -15733.607} C_VEL
LIN {X 0,Y 321.588,Z 480.157,A -85,B 0,C 180,E1 -15734.341,E2 -15734.341} C_VEL
LIN {X 0,Y 322.85,Z 431.133,A -85,B 0,C 180,E1 -15735.5,E2 -15735.5} C_VEL
LIN {X 0,Y 319.981,Z 416.77,A -85,B 0,C 180,E1 -15736.062,E2 -15736.062} C_VEL
LIN {X 0,Y 314.239,Z 400.394,A -85,B 0,C 180,E1 -15736.911,E2 -15736.911} C_VEL
LIN {X 0,Y 312.735,Z 392.53,A -85,B 0,C 180,E1 -15739.56,E2 -15739.56} C_VEL
LIN {X 0,Y 312.819,Z 392.521,A -85,B 0,C 180,E1 -15742.251,E2 -15742.251} C_VEL
LIN {X 0,Y 312.711,Z 392.532,A -85,B 0,C 180,E1 -15744.841,E2 -15744.841} C_VEL
LIN {X 0,Y 312.992,Z 392.497,A -85,B 0,C 180,E1 -15748.712,E2 -15748.712} C_VEL
LIN {X 0,Y 312.994,Z 392.495,A -85,B 0,C 180,E1 -15751.285,E2 -15751.285} C_VEL
LIN {X 0,Y 312.721,Z 392.528,A -85,B 0,C 180,E1 -15755.156,E2 -15755.156} C_VEL
LIN {X 0,Y 312.874,Z 392.51,A -85,B 0,C 180,E1 -15757.744,E2 -15757.744} C_VEL
LIN {X 0,Y 312.671,Z 392.536,A -85,B 0,C 180,E1 -15761.669,E2 -15761.669} C_VEL
LIN {X 0,Y 312.7,Z 392.531,A -85,B 0,C 180,E1 -15764.886,E2 -15764.886} C_VEL
LIN {X 0,Y 312.629,Z 392.538,A -85,B 0,C 180,E1 -15769.234,E2 -15769.234} C_VEL
LIN {X 0,Y 312.526,Z 392.553,A -85,B 0,C 180,E1 -15772.779,E2 -15772.779} C_VEL
LIN {X 0,Y 312.601,Z 392.545,A -85,B 0,C 180,E1 -15775.934,E2 -15775.934} C_VEL
LIN {X 0,Y 312.544,Z 392.552,A -85,B 0,C 180,E1 -15779.648,E2 -15779.648} C_VEL
LIN {X 0,Y 312.516,Z 392.559,A -85,B 0,C 180,E1 -15783.687,E2 -15783.687} C_VEL
LIN {X 0,Y 312.548,Z 392.553,A -85,B 0,C 180,E1 -15787.379,E2 -15787.379} C_VEL
LIN {X 0,Y 312.497,Z 392.556,A -85,B 0,C 180,E1 -15790.705,E2 -15790.705} C_VEL
LIN {X 0,Y 312.551,Z 392.652,A -85,B 0,C 180,E1 -15792.747,E2 -15792.747} C_VEL
LIN {X 0,Y 313.598,Z 397.919,A -85,B 0,C 180,E1 -15794.086,E2 -15794.086} C_VEL
LIN {X 0,Y 314.537,Z 399.267,A -85,B 0,C 180,E1 -15794.252,E2 -15794.252} C_VEL
LIN {X 0,Y 318.857,Z 404.956,A -85,B 0,C 180,E1 -15794.652,E2 -15794.652} C_VEL
LIN {X 0,Y 320.388,Z 408.81,A -85,B 0,C 180,E1 -15794.86,E2 -15794.86} C_VEL
LIN {X 0,Y 320.588,Z 412.552,A -85,B 0,C 180,E1 -15794.967,E2 -15794.967} C_VEL
LIN {X 0,Y 319.334,Z 416.474,A -85,B 0,C 180,E1 -15794.965,E2 -15794.965} C_VEL
LIN {X 0,Y 314.444,Z 425.285,A -85,B 0,C 180,E1 -15795.009,E2 -15795.009} C_VEL
LIN {X 0,Y 313.865,Z 428.608,A -85,B 0,C 180,E1 -15795.094,E2 -15795.094} C_VEL
LIN {X 0,Y 313.911,Z 429.164,A -85,B 0,C 180,E1 -15795.113,E2 -15795.113} C_VEL
LIN {X 0,Y 314.048,Z 434.996,A -85,B 0,C 180,E1 -15795.293,E2 -15795.293} C_VEL
LIN {X 0,Y 311.698,Z 509.036,A -85,B 0,C 180,E1 -15797.407,E2 -15797.407} C_VEL
LIN {X 0,Y 311.066,Z 522.118,A -85,B 0,C 180,E1 -15798.039,E2 -15798.039} C_VEL
LIN {X 0,Y 310.21,Z 535.025,A -85,B 0,C 180,E1 -15798.927,E2 -15798.927} C_VEL
LIN {X 0,Y 309.223,Z 547.309,A -85,B 0,C 180,E1 -15800.054,E2 -15800.054} C_VEL
LIN {X 0,Y 308.171,Z 558.529,A -85,B 0,C 180,E1 -15801.369,E2 -15801.369} C_VEL
LIN {X 0,Y 307.132,Z 568.926,A -85,B 0,C 180,E1 -15802.884,E2 -15802.884} C_VEL
LIN {X 0,Y 306.122,Z 578.258,A -85,B 0,C 180,E1 -15804.571,E2 -15804.571} C_VEL
LIN {X 0,Y 305.311,Z 586.773,A -85,B 0,C 180,E1 -15806.464,E2 -15806.464} C_VEL
LIN {X 0,Y 304.554,Z 594.458,A -85,B 0,C 180,E1 -15808.626,E2 -15808.626} C_VEL
LIN {X 0,Y 304.016,Z 600.876,A -85,B 0,C 180,E1 -15810.957,E2 -15810.957} C_VEL
LIN {X 0,Y 303.677,Z 605.374,A -85,B 0,C 180,E1 -15813.173,E2 -15813.173} C_VEL
LIN {X 0,Y 303.39,Z 608.5,A -85,B 0,C 180,E1 -15815.356,E2 -15815.356} C_VEL
LIN {X 0,Y 303.284,Z 609.928,A -85,B 0,C 180,E1 -15816.8,E2 -15816.8} C_VEL
LIN {X 0,Y 303.319,Z 610.798,A -85,B 0,C 180,E1 -15818.239,E2 -15818.239} C_VEL
LIN {X 0,Y 303.364,Z 611.193,A -85,B 0,C 180,E1 -15819.665,E2 -15819.665} C_VEL
LIN {X 0,Y 303.62,Z 610.925,A -85,B 0,C 180,E1 -15821.623,E2 -15821.623} C_VEL
LIN {X 0,Y 303.999,Z 609.483,A -85,B 0,C 180,E1 -15823.893,E2 -15823.893} C_VEL
LIN {X 0,Y 304.479,Z 607.286,A -85,B 0,C 180,E1 -15825.791,E2 -15825.791} C_VEL
LIN {X 0,Y 305.371,Z 603.496,A -85,B 0,C 180,E1 -15828.045,E2 -15828.045} C_VEL
LIN {X 0,Y 306.58,Z 598.214,A -85,B 0,C 180,E1 -15830.295,E2 -15830.295} C_VEL
LIN {X 0,Y 308.071,Z 591.557,A -85,B 0,C 180,E1 -15832.462,E2 -15832.462} C_VEL
LIN {X 0,Y 309.825,Z 583.639,A -85,B 0,C 180,E1 -15834.468,E2 -15834.468} C_VEL
LIN {X 0,Y 311.465,Z 575.579,A -85,B 0,C 180,E1 -15836.118,E2 -15836.118} C_VEL
LIN {X 0,Y 313.417,Z 565.802,A -85,B 0,C 180,E1 -15837.751,E2 -15837.751} C_VEL
LIN {X 0,Y 315.406,Z 554.473,A -85,B 0,C 180,E1 -15839.25,E2 -15839.25} C_VEL
LIN {X 0,Y 317.116,Z 543.353,A -85,B 0,C 180,E1 -15840.418,E2 -15840.418} C_VEL
LIN {X 0,Y 318.641,Z 531.016,A -85,B 0,C 180,E1 -15841.422,E2 -15841.422} C_VEL
LIN {X 0,Y 320.03,Z 517.173,A -85,B 0,C 180,E1 -15842.242,E2 -15842.242} C_VEL
LIN {X 0,Y 321.003,Z 502.97,A -85,B 0,C 180,E1 -15842.784,E2 -15842.784} C_VEL
LIN {X 0,Y 324.741,Z 435.776,A -85,B 0,C 180,E1 -15844.816,E2 -15844.816} C_VEL
LIN {X 0,Y 323.76,Z 430.746,A -85,B 0,C 180,E1 -15845.148,E2 -15845.148} C_VEL
LIN {X 0,Y 319.445,Z 421.03,A -85,B 0,C 180,E1 -15846.167,E2 -15846.167} C_VEL
LIN {X 0,Y 312.838,Z 408.345,A -85,B 0,C 180,E1 -15847.774,E2 -15847.774} C_VEL
LIN {X 0,Y 310.181,Z 403.923,A -85,B 0,C 180,E1 -15848.452,E2 -15848.452} C_VEL
LIN {X 0,Y 308.112,Z 400.38,A -85,B 0,C 180,E1 -15849.017,E2 -15849.017} C_VEL
LIN {X 0,Y 305.616,Z 393.416,A -85,B 0,C 180,E1 -15851.692,E2 -15851.692} C_VEL
LIN {X 0,Y 305.627,Z 393.417,A -85,B 0,C 180,E1 -15855.036,E2 -15855.036} C_VEL
LIN {X 0,Y 305.604,Z 393.418,A -85,B 0,C 180,E1 -15859.466,E2 -15859.466} C_VEL
LIN {X 0,Y 305.545,Z 393.423,A -85,B 0,C 180,E1 -15863.071,E2 -15863.071} C_VEL
LIN {X 0,Y 305.54,Z 393.425,A -85,B 0,C 180,E1 -15866.229,E2 -15866.229} C_VEL
LIN {X 0,Y 305.487,Z 393.434,A -85,B 0,C 180,E1 -15869.051,E2 -15869.051} C_VEL
LIN {X 0,Y 305.439,Z 393.438,A -85,B 0,C 180,E1 -15871.953,E2 -15871.953} C_VEL
LIN {X 0,Y 305.454,Z 393.435,A -85,B 0,C 180,E1 -15875.114,E2 -15875.114} C_VEL
LIN {X 0,Y 305.459,Z 393.435,A -85,B 0,C 180,E1 -15878.534,E2 -15878.534} C_VEL
LIN {X 0,Y 305.47,Z 393.433,A -85,B 0,C 180,E1 -15882.592,E2 -15882.592} C_VEL
LIN {X 0,Y 305.436,Z 393.437,A -85,B 0,C 180,E1 -15886.35,E2 -15886.35} C_VEL
LIN {X 0,Y 305.452,Z 393.437,A -85,B 0,C 180,E1 -15889.894,E2 -15889.894} C_VEL
LIN {X 0,Y 305.476,Z 393.433,A -85,B 0,C 180,E1 -15893.633,E2 -15893.633} C_VEL
LIN {X 0,Y 305.498,Z 393.528,A -85,B 0,C 180,E1 -15896.765,E2 -15896.765} C_VEL
LIN {X 0,Y 306.044,Z 395.428,A -85,B 0,C 180,E1 -15897.178,E2 -15897.178} C_VEL
LIN {X 0,Y 307.77,Z 398.453,A -85,B 0,C 180,E1 -15897.969,E2 -15897.969} C_VEL
LIN {X 0,Y 310.546,Z 406.763,A -85,B 0,C 180,E1 -15899.537,E2 -15899.537} C_VEL
LIN {X 0,Y 314.79,Z 416.356,A -85,B 0,C 180,E1 -15900.7,E2 -15900.7} C_VEL
LIN {X 0,Y 318.463,Z 425.653,A -85,B 0,C 180,E1 -15901.671,E2 -15901.671} C_VEL
LIN {X 0,Y 321.054,Z 440.599,A -85,B 0,C 180,E1 -15902.67,E2 -15902.67} C_VEL
LIN {X 0,Y 322.646,Z 452.991,A -85,B 0,C 180,E1 -15903.375,E2 -15903.375} C_VEL
LIN {X 0,Y 323.117,Z 460.292,A -85,B 0,C 180,E1 -15903.723,E2 -15903.723} C_VEL
LIN {X 0,Y 319.518,Z 526.008,A -85,B 0,C 180,E1 -15905.775,E2 -15905.775} C_VEL
LIN {X 0,Y 318.217,Z 539.152,A -85,B 0,C 180,E1 -15906.405,E2 -15906.405} C_VEL
LIN {X 0,Y 316.789,Z 550.395,A -85,B 0,C 180,E1 -15907.157,E2 -15907.157} C_VEL
LIN {X 0,Y 315.021,Z 562.442,A -85,B 0,C 180,E1 -15908.231,E2 -15908.231} C_VEL
LIN {X 0,Y 313.13,Z 573.414,A -85,B 0,C 180,E1 -15909.472,E2 -15909.472} C_VEL
LIN {X 0,Y 311.316,Z 583.458,A -85,B 0,C 180,E1 -15910.895,E2 -15910.895} C_VEL
LIN {X 0,Y 309.62,Z 592.279,A -85,B 0,C 180,E1 -15912.431,E2 -15912.431} C_VEL
LIN {X 0,Y 307.877,Z 601.566,A -85,B 0,C 180,E1 -15914.443,E2 -15914.443} C_VEL
LIN {X 0,Y 306.393,Z 608.777,A -85,B 0,C 180,E1 -15916.404,E2 -15916.404} C_VEL
LIN {X 0,Y 305.386,Z 613.698,A -85,B 0,C 180,E1 -15918.048,E2 -15918.048} C_VEL
LIN {X 0,Y 304.564,Z 618.456,A -85,B 0,C 180,E1 -15920.036,E2 -15920.036} C_VEL
LIN {X 0,Y 304.012,Z 622.073,A -85,B 0,C 180,E1 -15922.029,E2 -15922.029} C_VEL
LIN {X 0,Y 303.694,Z 624.927,A -85,B 0,C 180,E1 -15924.323,E2 -15924.323} C_VEL
LIN {X 0,Y 303.607,Z 627.206,A -85,B 0,C 180,E1 -15927.348,E2 -15927.348} C_VEL
LIN {X 0,Y 303.575,Z 628.074,A -85,B 0,C 180,E1 -15928.675,E2 -15928.675} C_VEL
LIN {X 0,Y 303.603,Z 628.495,A -85,B 0,C 180,E1 -15930.002,E2 -15930.002} C_VEL
LIN {X 0,Y 303.565,Z 628.507,A -85,B 0,C 180,E1 -15931.328,E2 -15931.328} C_VEL
LIN {X 0,Y 303.602,Z 628.127,A -85,B 0,C 180,E1 -15932.655,E2 -15932.655} C_VEL
LIN {X 0,Y 303.593,Z 627.35,A -85,B 0,C 180,E1 -15933.984,E2 -15933.984} C_VEL
LIN {X 0,Y 303.626,Z 625.862,A -85,B 0,C 180,E1 -15935.546,E2 -15935.546} C_VEL
LIN {X 0,Y 303.994,Z 622.423,A -85,B 0,C 180,E1 -15937.975,E2 -15937.975} C_VEL
LIN {X 0,Y 304.501,Z 618.448,A -85,B 0,C 180,E1 -15939.97,E2 -15939.97} C_VEL
LIN {X 0,Y 305.315,Z 613.341,A -85,B 0,C 180,E1 -15941.958,E2 -15941.958} C_VEL
LIN {X 0,Y 306.527,Z 606.945,A -85,B 0,C 180,E1 -15943.932,E2 -15943.932} C_VEL
LIN {X 0,Y 307.963,Z 598.958,A -85,B 0,C 180,E1 -15945.895,E2 -15945.895} C_VEL
LIN {X 0,Y 309.305,Z 591.03,A -85,B 0,C 180,E1 -15947.489,E2 -15947.489} C_VEL
LIN {X 0,Y 311.032,Z 580.986,A -85,B 0,C 180,E1 -15949.127,E2 -15949.127} C_VEL
LIN {X 0,Y 312.843,Z 569.997,A -85,B 0,C 180,E1 -15950.551,E2 -15950.551} C_VEL
LIN {X 0,Y 314.658,Z 557.534,A -85,B 0,C 180,E1 -15951.799,E2 -15951.799} C_VEL
LIN {X 0,Y 315.94,Z 546.512,A -85,B 0,C 180,E1 -15952.652,E2 -15952.652} C_VEL
LIN {X 0,Y 317.128,Z 534.523,A -85,B 0,C 180,E1 -15953.338,E2 -15953.338} C_VEL
LIN {X 0,Y 318.034,Z 521.078,A -85,B 0,C 180,E1 -15953.839,E2 -15953.839} C_VEL
LIN {X 0,Y 320.004,Z 458.241,A -85,B 0,C 180,E1 -15955.402,E2 -15955.402} C_VEL
LIN {X 0,Y 316.981,Z 438.313,A -85,B 0,C 180,E1 -15956.283,E2 -15956.283} C_VEL
LIN {X 0,Y 313.688,Z 422.947,A -85,B 0,C 180,E1 -15957.088,E2 -15957.088} C_VEL
LIN {X 0,Y 310.458,Z 415.309,A -85,B 0,C 180,E1 -15957.719,E2 -15957.719} C_VEL
LIN {X 0,Y 309.002,Z 407.989,A -85,B 0,C 180,E1 -15960.199,E2 -15960.199} C_VEL
LIN {X 0,Y 306.972,Z 399.342,A -85,B 0,C 180,E1 -15963.332,E2 -15963.332} C_VEL
LIN {X 0,Y 305.488,Z 393.434,A -85,B 0,C 180,E1 -15965.617,E2 -15965.617} C_VEL
LIN {X 0,Y 305.472,Z 393.438,A -85,B 0,C 180,E1 -15968.534,E2 -15968.534} C_VEL
LIN {X 0,Y 305.46,Z 393.437,A -85,B 0,C 180,E1 -15972.587,E2 -15972.587} C_VEL
LIN {X 0,Y 305.431,Z 393.441,A -85,B 0,C 180,E1 -15976.346,E2 -15976.346} C_VEL
LIN {X 0,Y 305.464,Z 393.429,A -85,B 0,C 180,E1 -15979.893,E2 -15979.893} C_VEL
LIN {X 0,Y 305.487,Z 393.43,A -85,B 0,C 180,E1 -15983.632,E2 -15983.632} C_VEL
LIN {X 0,Y 305.471,Z 393.427,A -85,B 0,C 180,E1 -15986.484,E2 -15986.484} C_VEL
LIN {X 0,Y 305.464,Z 393.425,A -85,B 0,C 180,E1 -15989.591,E2 -15989.591} C_VEL
LIN {X 0,Y 305.521,Z 393.422,A -85,B 0,C 180,E1 -15992.609,E2 -15992.609} C_VEL
LIN {X 0,Y 305.514,Z 393.428,A -85,B 0,C 180,E1 -15995.539,E2 -15995.539} C_VEL
LIN {X 0,Y 305.527,Z 393.427,A -85,B 0,C 180,E1 -15999.816,E2 -15999.816} C_VEL
LIN {X 0,Y 305.581,Z 393.417,A -85,B 0,C 180,E1 -16002.603,E2 -16002.603} C_VEL
LIN {X 0,Y 305.656,Z 393.4,A -85,B 0,C 180,E1 -16005.349,E2 -16005.349} C_VEL
LIN {X 0,Y 305.645,Z 393.402,A -85,B 0,C 180,E1 -16009.4,E2 -16009.4} C_VEL
LIN {X 0,Y 305.82,Z 393.39,A -85,B 0,C 180,E1 -16012.075,E2 -16012.075} C_VEL
LIN {X 0,Y 305.695,Z 393.407,A -85,B 0,C 180,E1 -16014.724,E2 -16014.724} C_VEL
LIN {X 0,Y 305.962,Z 393.374,A -85,B 0,C 180,E1 -16018.684,E2 -16018.684} C_VEL
LIN {X 0,Y 305.962,Z 393.369,A -85,B 0,C 180,E1 -16021.316,E2 -16021.316} C_VEL
LIN {X 0,Y 305.858,Z 393.381,A -85,B 0,C 180,E1 -16026.609,E2 -16026.609} C_VEL
LIN {X 0,Y 305.743,Z 393.398,A -85,B 0,C 180,E1 -16029.26,E2 -16029.26} C_VEL
LIN {X 0,Y 305.596,Z 393.421,A -85,B 0,C 180,E1 -16033.296,E2 -16033.296} C_VEL
LIN {X 0,Y 305.601,Z 393.417,A -85,B 0,C 180,E1 -16036.02,E2 -16036.02} C_VEL
LIN {X 0,Y 305.599,Z 393.42,A -85,B 0,C 180,E1 -16039.453,E2 -16039.453} C_VEL
LIN {X 0,Y 305.547,Z 393.569,A -85,B 0,C 180,E1 -16040.535,E2 -16040.535} C_VEL
LIN {X 0,Y 307.609,Z 402.113,A -85,B 0,C 180,E1 -16044.039,E2 -16044.039} C_VEL
LIN {X 0,Y 315.746,Z 419.238,A -85,B 0,C 180,E1 -16045.503,E2 -16045.503} C_VEL
LIN {X 0,Y 319.669,Z 429.153,A -85,B 0,C 180,E1 -16046.208,E2 -16046.208} C_VEL
LIN {X 0,Y 320.694,Z 434.192,A -85,B 0,C 180,E1 -16046.457,E2 -16046.457} C_VEL
LIN {X 0,Y 318.172,Z 509.096,A -85,B 0,C 180,E1 -16048.336,E2 -16048.336} C_VEL
LIN {X 0,Y 317.35,Z 521.471,A -85,B 0,C 180,E1 -16048.868,E2 -16048.868} C_VEL
LIN {X 0,Y 316.108,Z 534.674,A -85,B 0,C 180,E1 -16049.7,E2 -16049.7} C_VEL
LIN {X 0,Y 314.694,Z 546.777,A -85,B 0,C 180,E1 -16050.757,E2 -16050.757} C_VEL
LIN {X 0,Y 313.041,Z 558.547,A -85,B 0,C 180,E1 -16052.087,E2 -16052.087} C_VEL
LIN {X 0,Y 311.549,Z 567.953,A -85,B 0,C 180,E1 -16053.418,E2 -16053.418} C_VEL
LIN {X 0,Y 310.085,Z 576.26,A -85,B 0,C 180,E1 -16054.848,E2 -16054.848} C_VEL
LIN {X 0,Y 308.392,Z 584.874,A -85,B 0,C 180,E1 -16056.666,E2 -16056.666} C_VEL
LIN {X 0,Y 306.824,Z 593.034,A -85,B 0,C 180,E1 -16058.848,E2 -16058.848} C_VEL
LIN {X 0,Y 305.851,Z 598.454,A -85,B 0,C 180,E1 -16060.684,E2 -16060.684} C_VEL
LIN {X 0,Y 305.039,Z 602.748,A -85,B 0,C 180,E1 -16062.499,E2 -16062.499} C_VEL
LIN {X 0,Y 304.422,Z 606.089,A -85,B 0,C 180,E1 -16064.299,E2 -16064.299} C_VEL
LIN {X 0,Y 303.979,Z 608.583,A -85,B 0,C 180,E1 -16066.082,E2 -16066.082} C_VEL
LIN {X 0,Y 303.61,Z 610.26,A -85,B 0,C 180,E1 -16067.831,E2 -16067.831} C_VEL
LIN {X 0,Y 303.384,Z 611.315,A -85,B 0,C 180,E1 -16069.859,E2 -16069.859} C_VEL
LIN {X 0,Y 303.282,Z 611.417,A -85,B 0,C 180,E1 -16071.989,E2 -16071.989} C_VEL
LIN {X 0,Y 303.4,Z 610.119,A -85,B 0,C 180,E1 -16074.611,E2 -16074.611} C_VEL
LIN {X 0,Y 303.73,Z 607.302,A -85,B 0,C 180,E1 -16077.152,E2 -16077.152} C_VEL
LIN {X 0,Y 304.224,Z 603.375,A -85,B 0,C 180,E1 -16079.452,E2 -16079.452} C_VEL
LIN {X 0,Y 304.889,Z 597.494,A -85,B 0,C 180,E1 -16081.906,E2 -16081.906} C_VEL
LIN {X 0,Y 305.803,Z 590.57,A -85,B 0,C 180,E1 -16084.107,E2 -16084.107} C_VEL
LIN {X 0,Y 306.823,Z 582.921,A -85,B 0,C 180,E1 -16086.025,E2 -16086.025} C_VEL
LIN {X 0,Y 308.105,Z 573.62,A -85,B 0,C 180,E1 -16087.889,E2 -16087.889} C_VEL
LIN {X 0,Y 309.501,Z 563.198,A -85,B 0,C 180,E1 -16089.564,E2 -16089.564} C_VEL
LIN {X 0,Y 310.809,Z 551.465,A -85,B 0,C 180,E1 -16091.048,E2 -16091.048} C_VEL
LIN {X 0,Y 312.052,Z 539.657,A -85,B 0,C 180,E1 -16092.213,E2 -16092.213} C_VEL
LIN {X 0,Y 312.976,Z 527.885,A -85,B 0,C 180,E1 -16093.098,E2 -16093.098} C_VEL
LIN {X 0,Y 313.842,Z 514.123,A -85,B 0,C 180,E1 -16093.83,E2 -16093.83} C_VEL
LIN {X 0,Y 314.363,Z 501.436,A -85,B 0,C 180,E1 -16094.251,E2 -16094.251} C_VEL
LIN {X 0,Y 316.178,Z 431.959,A -85,B 0,C 180,E1 -16095.928,E2 -16095.928} C_VEL
LIN {X 0,Y 313.588,Z 419.017,A -85,B 0,C 180,E1 -16096.45,E2 -16096.45} C_VEL
LIN {X 0,Y 307.034,Z 400.587,A -85,B 0,C 180,E1 -16097.438,E2 -16097.438} C_VEL
LIN {X 0,Y 305.684,Z 393.409,A -85,B 0,C 180,E1 -16099.985,E2 -16099.985} C_VEL
LIN {X 0,Y 305.801,Z 393.391,A -85,B 0,C 180,E1 -16103.4,E2 -16103.4} C_VEL
LIN {X 0,Y 305.888,Z 393.38,A -85,B 0,C 180,E1 -16107.365,E2 -16107.365} C_VEL
LIN {X 0,Y 306.058,Z 393.361,A -85,B 0,C 180,E1 -16109.998,E2 -16109.998} C_VEL
LIN {X 0,Y 305.89,Z 393.38,A -85,B 0,C 180,E1 -16112.632,E2 -16112.632} C_VEL
LIN {X 0,Y 305.855,Z 393.384,A -85,B 0,C 180,E1 -16116.596,E2 -16116.596} C_VEL
LIN {X 0,Y 305.737,Z 393.399,A -85,B 0,C 180,E1 -16119.258,E2 -16119.258} C_VEL
LIN {X 0,Y 305.59,Z 393.416,A -85,B 0,C 180,E1 -16123.294,E2 -16123.294} C_VEL
LIN {X 0,Y 305.595,Z 393.422,A -85,B 0,C 180,E1 -16126.018,E2 -16126.018} C_VEL
LIN {X 0,Y 305.575,Z 393.417,A -85,B 0,C 180,E1 -16129.443,E2 -16129.443} C_VEL
LIN {X 0,Y 305.484,Z 393.43,A -85,B 0,C 180,E1 -16133.037,E2 -16133.037} C_VEL
LIN {X 0,Y 305.546,Z 393.421,A -85,B 0,C 180,E1 -16136.225,E2 -16136.225} C_VEL
LIN {X 0,Y 305.494,Z 393.426,A -85,B 0,C 180,E1 -16139.048,E2 -16139.048} C_VEL
LIN {X 0,Y 305.445,Z 393.438,A -85,B 0,C 180,E1 -16141.95,E2 -16141.95} C_VEL
LIN {X 0,Y 305.459,Z 393.434,A -85,B 0,C 180,E1 -16145.111,E2 -16145.111} C_VEL
LIN {X 0,Y 305.487,Z 393.43,A -85,B 0,C 180,E1 -16148.537,E2 -16148.537} C_VEL
LIN {X 0,Y 305.504,Z 393.491,A -85,B 0,C 180,E1 -16152.481,E2 -16152.481} C_VEL
LIN {X 0,Y 306.467,Z 398.408,A -85,B 0,C 180,E1 -16153.75,E2 -16153.75} C_VEL
LIN {X 0,Y 311.595,Z 415.383,A -85,B 0,C 180,E1 -16154.573,E2 -16154.573} C_VEL
LIN {X 0,Y 313.911,Z 429.164,A -85,B 0,C 180,E1 -16155.113,E2 -16155.113} C_VEL
LIN {X 0,Y 313.959,Z 433.018,A -85,B 0,C 180,E1 -16155.229,E2 -16155.229} C_VEL
LIN {X 0,Y 313.292,Z 436.86,A -85,B 0,C 180,E1 -16155.307,E2 -16155.307} C_VEL
LIN {X 0,Y 310.74,Z 444.382,A -85,B 0,C 180,E1 -16155.4,E2 -16155.4} C_VEL
LIN {X 0,Y 307.327,Z 453.845,A -85,B 0,C 180,E1 -16155.509,E2 -16155.509} C_VEL
LIN {X 0,Y 306.451,Z 459.715,A -85,B 0,C 180,E1 -16155.644,E2 -16155.644} C_VEL
LIN {X 0,Y 304.79,Z 509.495,A -85,B 0,C 180,E1 -16157.12,E2 -16157.12} C_VEL
LIN {X 0,Y 304.122,Z 522.487,A -85,B 0,C 180,E1 -16157.769,E2 -16157.769} C_VEL
LIN {X 0,Y 303.156,Z 536.312,A -85,B 0,C 180,E1 -16158.756,E2 -16158.756} C_VEL
LIN {X 0,Y 302.097,Z 548.88,A -85,B 0,C 180,E1 -16159.973,E2 -16159.973} C_VEL
LIN {X 0,Y 301.026,Z 560.095,A -85,B 0,C 180,E1 -16161.352,E2 -16161.352} C_VEL
LIN {X 0,Y 299.914,Z 570.921,A -85,B 0,C 180,E1 -16163.033,E2 -16163.033} C_VEL
LIN {X 0,Y 298.882,Z 580.196,A -85,B 0,C 180,E1 -16164.807,E2 -16164.807} C_VEL
LIN {X 0,Y 298.077,Z 588.376,A -85,B 0,C 180,E1 -16166.757,E2 -16166.757} C_VEL
LIN {X 0,Y 297.352,Z 596.071,A -85,B 0,C 180,E1 -16169.065,E2 -16169.065} C_VEL
LIN {X 0,Y 296.884,Z 601.436,A -85,B 0,C 180,E1 -16171.145,E2 -16171.145} C_VEL
LIN {X 0,Y 296.586,Z 605.56,A -85,B 0,C 180,E1 -16173.241,E2 -16173.241} C_VEL
LIN {X 0,Y 296.376,Z 607.8,A -85,B 0,C 180,E1 -16174.733,E2 -16174.733} C_VEL
LIN {X 0,Y 296.223,Z 609.473,A -85,B 0,C 180,E1 -16176.213,E2 -16176.213} C_VEL
LIN {X 0,Y 296.182,Z 610.64,A -85,B 0,C 180,E1 -16177.725,E2 -16177.725} C_VEL
LIN {X 0,Y 296.237,Z 611.278,A -85,B 0,C 180,E1 -16179.153,E2 -16179.153} C_VEL
LIN {X 0,Y 296.492,Z 611.269,A -85,B 0,C 180,E1 -16181.462,E2 -16181.462} C_VEL
LIN {X 0,Y 296.808,Z 610.278,A -85,B 0,C 180,E1 -16183.492,E2 -16183.492} C_VEL
LIN {X 0,Y 297.37,Z 608.128,A -85,B 0,C 180,E1 -16185.685,E2 -16185.685} C_VEL
LIN {X 0,Y 298.15,Z 605.038,A -85,B 0,C 180,E1 -16187.752,E2 -16187.752} C_VEL
LIN {X 0,Y 299.486,Z 599.767,A -85,B 0,C 180,E1 -16190.254,E2 -16190.254} C_VEL
LIN {X 0,Y 300.885,Z 594.066,A -85,B 0,C 180,E1 -16192.281,E2 -16192.281} C_VEL
LIN {X 0,Y 302.61,Z 586.767,A -85,B 0,C 180,E1 -16194.335,E2 -16194.335} C_VEL
LIN {X 0,Y 304.678,Z 577.704,A -85,B 0,C 180,E1 -16196.363,E2 -16196.363} C_VEL
LIN {X 0,Y 306.871,Z 567.24,A -85,B 0,C 180,E1 -16198.195,E2 -16198.195} C_VEL
LIN {X 0,Y 308.948,Z 556.357,A -85,B 0,C 180,E1 -16199.707,E2 -16199.707} C_VEL
LIN {X 0,Y 310.896,Z 544.404,A -85,B 0,C 180,E1 -16201.013,E2 -16201.013} C_VEL
LIN {X 0,Y 312.627,Z 531.627,A -85,B 0,C 180,E1 -16202.093,E2 -16202.093} C_VEL
LIN {X 0,Y 314.104,Z 518.06,A -85,B 0,C 180,E1 -16202.926,E2 -16202.926} C_VEL
LIN {X 0,Y 315.095,Z 504.608,A -85,B 0,C 180,E1 -16203.476,E2 -16203.476} C_VEL
LIN {X 0,Y 319.119,Z 437.249,A -85,B 0,C 180,E1 -16205.547,E2 -16205.547} C_VEL
LIN {X 0,Y 318.324,Z 433.569,A -85,B 0,C 180,E1 -16205.819,E2 -16205.819} C_VEL
LIN {X 0,Y 314.414,Z 424.786,A -85,B 0,C 180,E1 -16206.8,E2 -16206.8} C_VEL
LIN {X 0,Y 308.35,Z 412.803,A -85,B 0,C 180,E1 -16208.376,E2 -16208.376} C_VEL
LIN {X 0,Y 303.487,Z 404.836,A -85,B 0,C 180,E1 -16209.677,E2 -16209.677} C_VEL
LIN {X 0,Y 300.881,Z 400.647,A -85,B 0,C 180,E1 -16210.451,E2 -16210.451} C_VEL
LIN {X 0,Y 298.552,Z 394.296,A -85,B 0,C 180,E1 -16213.009,E2 -16213.009} C_VEL
LIN {X 0,Y 298.539,Z 394.299,A -85,B 0,C 180,E1 -16216.409,E2 -16216.409} C_VEL
LIN {X 0,Y 298.555,Z 394.295,A -85,B 0,C 180,E1 -16219.684,E2 -16219.684} C_VEL
LIN {X 0,Y 298.48,Z 394.306,A -85,B 0,C 180,E1 -16223.596,E2 -16223.596} C_VEL
LIN {X 0,Y 298.48,Z 394.305,A -85,B 0,C 180,E1 -16226.575,E2 -16226.575} C_VEL
